LIN {X 0,Y 290.074,Z 393.623,A -85,B 0,C 180,E1 -16659.764,E2 -16659.764} C_VEL
LIN {X 0,Y 290.99,Z 387.907,A -85,B 0,C 180,E1 -16662.554,E2 -16662.554} C_VEL
LIN {X 0,Y 292.274,Z 381.468,A -85,B 0,C 180,E1 -16664.981,E2 -16664.981} C_VEL
LIN {X 0,Y 293.884,Z 373.47,A -85,B 0,C 180,E1 -16667.393,E2 -16667.393} C_VEL
LIN {X 0,Y 295.651,Z 365.107,A -85,B 0,C 180,E1 -16669.439,E2 -16669.439} C_VEL
LIN {X 0,Y 297.748,Z 355.042,A -85,B 0,C 180,E1 -16671.46,E2 -16671.46} C_VEL
LIN {X 0,Y 300.058,Z 343.813,A -85,B 0,C 180,E1 -16673.281,E2 -16673.281} C_VEL
LIN {X 0,Y 302.413,Z 331.182,A -85,B 0,C 180,E1 -16674.916,E2 -16674.916} C_VEL
LIN {X 0,Y 303.356,Z 325.276,A -85,B 0,C 180,E1 -16675.567,E2 -16675.567} C_VEL
LIN {X 0,Y 302.15,Z 313.202,A -85,B 0,C 180,E1 -16676.964,E2 -16676.964} C_VEL
LIN {X 0,Y 300.276,Z 302.153,A -85,B 0,C 180,E1 -16678.11,E2 -16678.11} C_VEL
LIN {X 0,Y 297.094,Z 288.461,A -85,B 0,C 180,E1 -16679.359,E2 -16679.359} C_VEL
LIN {X 0,Y 292.982,Z 275.551,A -85,B 0,C 180,E1 -16680.427,E2 -16680.427} C_VEL
LIN {X 0,Y 291.562,Z 271.297,A -85,B 0,C 180,E1 -16680.732,E2 -16680.732} C_VEL
LIN {X 0,Y 291.469,Z 270.609,A -85,B 0,C 180,E1 -16680.823,E2 -16680.823} C_VEL
LIN {X 0,Y 292.181,Z 265.371,A -85,B 0,C 180,E1 -16685.26,E2 -16685.26} C_VEL
LIN {X 0,Y 292.643,Z 261.551,A -85,B 0,C 180,E1 -16688.639,E2 -16688.639} C_VEL
LIN {X 0,Y 292.591,Z 258.142,A -85,B 0,C 180,E1 -16691.874,E2 -16691.874} C_VEL
LIN {X 0,Y 292.078,Z 254.325,A -85,B 0,C 180,E1 -16695.749,E2 -16695.749} C_VEL
LIN {X 0,Y 291.598,Z 250.967,A -85,B 0,C 180,E1 -16699.402,E2 -16699.402} C_VEL
LIN {X 0,Y 291.376,Z 249.818,A -85,B 0,C 180,E1 -16700.835,E2 -16700.835} C_VEL
LIN {X 0,Y 291.362,Z 249.821,A -85,B 0,C 180,E1 -16704.626,E2 -16704.626} C_VEL
LIN {X 0,Y 291.366,Z 249.819,A -85,B 0,C 180,E1 -16707.95,E2 -16707.95} C_VEL
LIN {X 0,Y 291.345,Z 249.821,A -85,B 0,C 180,E1 -16711.154,E2 -16711.154} C_VEL
LIN {X 0,Y 291.36,Z 249.818,A -85,B 0,C 180,E1 -16714.267,E2 -16714.267} C_VEL
LIN {X 0,Y 291.372,Z 249.817,A -85,B 0,C 180,E1 -16717.299,E2 -16717.299} C_VEL
LIN {X 0,Y 291.459,Z 249.806,A -85,B 0,C 180,E1 -16720.27,E2 -16720.27} C_VEL
LIN {X 0,Y 291.515,Z 249.797,A -85,B 0,C 180,E1 -16724.653,E2 -16724.653} C_VEL
LIN {X 0,Y 291.53,Z 249.79,A -85,B 0,C 180,E1 -16728.88,E2 -16728.88} C_VEL
LIN {X 0,Y 291.653,Z 249.782,A -85,B 0,C 180,E1 -16731.687,E2 -16731.687} C_VEL
LIN {X 0,Y 291.608,Z 249.785,A -85,B 0,C 180,E1 -16734.468,E2 -16734.468} C_VEL
LIN {X 0,Y 291.89,Z 249.751,A -85,B 0,C 180,E1 -16738.62,E2 -16738.62} C_VEL
LIN {X 0,Y 291.885,Z 249.752,A -85,B 0,C 180,E1 -16741.38,E2 -16741.38} C_VEL
LIN {X 0,Y 291.737,Z 249.77,A -85,B 0,C 180,E1 -16746.918,E2 -16746.918} C_VEL
LIN {X 0,Y 291.577,Z 249.791,A -85,B 0,C 180,E1 -16749.714,E2 -16749.714} C_VEL
LIN {X 0,Y 291.524,Z 249.795,A -85,B 0,C 180,E1 -16753.95,E2 -16753.95} C_VEL
LIN {X 0,Y 291.489,Z 249.801,A -85,B 0,C 180,E1 -16756.818,E2 -16756.818} C_VEL
LIN {X 0,Y 291.452,Z 249.804,A -85,B 0,C 180,E1 -16759.875,E2 -16759.875} C_VEL
LIN {X 0,Y 291.384,Z 249.814,A -85,B 0,C 180,E1 -16764.207,E2 -16764.207} C_VEL
LIN {X 0,Y 291.422,Z 249.81,A -85,B 0,C 180,E1 -16767.272,E2 -16767.272} C_VEL
LIN {X 0,Y 291.335,Z 249.821,A -85,B 0,C 180,E1 -16770.437,E2 -16770.437} C_VEL
LIN {X 0,Y 291.346,Z 249.82,A -85,B 0,C 180,E1 -16773.698,E2 -16773.698} C_VEL
LIN {X 0,Y 291.36,Z 249.818,A -85,B 0,C 180,E1 -16777.25,E2 -16777.25} C_VEL
LIN {X 0,Y 291.301,Z 249.828,A -85,B 0,C 180,E1 -16780.648,E2 -16780.648} C_VEL
LIN {X 0,Y 291.291,Z 249.828,A -85,B 0,C 180,E1 -16784.402,E2 -16784.402} C_VEL
LIN {X 0,Y 291.298,Z 249.899,A -85,B 0,C 180,E1 -16785.6,E2 -16785.6} C_VEL
LIN {X 0,Y 291.68,Z 252.914,A -85,B 0,C 180,E1 -16789.416,E2 -16789.416} C_VEL
LIN {X 0,Y 291.669,Z 255.712,A -85,B 0,C 180,E1 -16792.671,E2 -16792.671} C_VEL
LIN {X 0,Y 291.365,Z 258.994,A -85,B 0,C 180,E1 -16796.304,E2 -16796.304} C_VEL
LIN {X 0,Y 291.017,Z 261.76,A -85,B 0,C 180,E1 -16799.228,E2 -16799.228} C_VEL
LIN {X 0,Y 292.207,Z 265.24,A -85,B 0,C 180,E1 -16799.504,E2 -16799.504} C_VEL
LIN {X 0,Y 297.427,Z 279.57,A -85,B 0,C 180,E1 -16800.774,E2 -16800.774} C_VEL
LIN {X 0,Y 301.068,Z 292.825,A -85,B 0,C 180,E1 -16802.074,E2 -16802.074} C_VEL
LIN {X 0,Y 303.481,Z 304.486,A -85,B 0,C 180,E1 -16803.353,E2 -16803.353} C_VEL
LIN {X 0,Y 304.465,Z 311.537,A -85,B 0,C 180,E1 -16804.19,E2 -16804.19} C_VEL
LIN {X 0,Y 302.688,Z 323.224,A -85,B 0,C 180,E1 -16805.479,E2 -16805.479} C_VEL
LIN {X 0,Y 300.437,Z 335.236,A -85,B 0,C 180,E1 -16807.114,E2 -16807.114} C_VEL
LIN {X 0,Y 298.279,Z 346.061,A -85,B 0,C 180,E1 -16808.942,E2 -16808.942} C_VEL
LIN {X 0,Y 296.117,Z 355.805,A -85,B 0,C 180,E1 -16810.953,E2 -16810.953} C_VEL
LIN {X 0,Y 294.307,Z 363.822,A -85,B 0,C 180,E1 -16812.972,E2 -16812.972} C_VEL
LIN {X 0,Y 293,Z 370.611,A -85,B 0,C 180,E1 -16815.057,E2 -16815.057} C_VEL
LIN {X 0,Y 291.561,Z 377.013,A -85,B 0,C 180,E1 -16817.471,E2 -16817.471} C_VEL
LIN {X 0,Y 290.543,Z 382.685,A -85,B 0,C 180,E1 -16820.252,E2 -16820.252} C_VEL
LIN {X 0,Y 289.89,Z 386.805,A -85,B 0,C 180,E1 -16823.038,E2 -16823.038} C_VEL
LIN {X 0,Y 289.58,Z 389.498,A -85,B 0,C 180,E1 -16825.825,E2 -16825.825} C_VEL
LIN {X 0,Y 289.4,Z 390.846,A -85,B 0,C 180,E1 -16828.609,E2 -16828.609} C_VEL
LIN {X 0,Y 289.4,Z 390.876,A -85,B 0,C 180,E1 -16831.392,E2 -16831.392} C_VEL
LIN {X 0,Y 289.579,Z 389.585,A -85,B 0,C 180,E1 -16834.176,E2 -16834.176} C_VEL
LIN {X 0,Y 289.89,Z 386.945,A -85,B 0,C 180,E1 -16836.963,E2 -16836.963} C_VEL
LIN {X 0,Y 290.53,Z 382.885,A -85,B 0,C 180,E1 -16839.749,E2 -16839.749} C_VEL
LIN {X 0,Y 291.502,Z 377.275,A -85,B 0,C 180,E1 -16842.532,E2 -16842.532} C_VEL
LIN {X 0,Y 292.955,Z 370.934,A -85,B 0,C 180,E1 -16844.945,E2 -16844.945} C_VEL
LIN {X 0,Y 294.134,Z 364.631,A -85,B 0,C 180,E1 -16846.917,E2 -16846.917} C_VEL
LIN {X 0,Y 296.005,Z 356.282,A -85,B 0,C 180,E1 -16849.054,E2 -16849.054} C_VEL
LIN {X 0,Y 298.156,Z 346.631,A -85,B 0,C 180,E1 -16851.068,E2 -16851.068} C_VEL
LIN {X 0,Y 300.327,Z 335.919,A -85,B 0,C 180,E1 -16852.895,E2 -16852.895} C_VEL
LIN {X 0,Y 302.591,Z 324.044,A -85,B 0,C 180,E1 -16854.53,E2 -16854.53} C_VEL
LIN {X 0,Y 304.434,Z 312.231,A -85,B 0,C 180,E1 -16855.849,E2 -16855.849} C_VEL
LIN {X 0,Y 304.028,Z 307.686,A -85,B 0,C 180,E1 -16856.38,E2 -16856.38} C_VEL
LIN {X 0,Y 301.698,Z 295.36,A -85,B 0,C 180,E1 -16857.769,E2 -16857.769} C_VEL
LIN {X 0,Y 298.177,Z 281.925,A -85,B 0,C 180,E1 -16859.117,E2 -16859.117} C_VEL
LIN {X 0,Y 293.385,Z 268.223,A -85,B 0,C 180,E1 -16860.363,E2 -16860.363} C_VEL
LIN {X 0,Y 291.091,Z 262.196,A -85,B 0,C 180,E1 -16860.852,E2 -16860.852} C_VEL
LIN {X 0,Y 291.063,Z 261.708,A -85,B 0,C 180,E1 -16860.948,E2 -16860.948} C_VEL
LIN {X 0,Y 291.509,Z 257.962,A -85,B 0,C 180,E1 -16864.944,E2 -16864.944} C_VEL
LIN {X 0,Y 291.722,Z 254.552,A -85,B 0,C 180,E1 -16868.784,E2 -16868.784} C_VEL
LIN {X 0,Y 291.606,Z 252.15,A -85,B 0,C 180,E1 -16871.657,E2 -16871.657} C_VEL
LIN {X 0,Y 291.309,Z 250.01,A -85,B 0,C 180,E1 -16874.399,E2 -16874.399} C_VEL
LIN {X 0,Y 291.29,Z 249.83,A -85,B 0,C 180,E1 -16877.502,E2 -16877.502} C_VEL
LIN {X 0,Y 291.336,Z 249.822,A -85,B 0,C 180,E1 -16881.155,E2 -16881.155} C_VEL
LIN {X 0,Y 291.357,Z 249.82,A -85,B 0,C 180,E1 -16884.625,E2 -16884.625} C_VEL
LIN {X 0,Y 291.373,Z 249.816,A -85,B 0,C 180,E1 -16887.951,E2 -16887.951} C_VEL
LIN {X 0,Y 291.38,Z 249.816,A -85,B 0,C 180,E1 -16891.158,E2 -16891.158} C_VEL
LIN {X 0,Y 291.418,Z 249.806,A -85,B 0,C 180,E1 -16894.272,E2 -16894.272} C_VEL
LIN {X 0,Y 291.377,Z 249.816,A -85,B 0,C 180,E1 -16897.299,E2 -16897.299} C_VEL
LIN {X 0,Y 291.461,Z 249.804,A -85,B 0,C 180,E1 -16900.27,E2 -16900.27} C_VEL
LIN {X 0,Y 291.558,Z 249.791,A -85,B 0,C 180,E1 -16904.624,E2 -16904.624} C_VEL
LIN {X 0,Y 291.532,Z 249.795,A -85,B 0,C 180,E1 -16908.88,E2 -16908.88} C_VEL
LIN {X 0,Y 291.553,Z 249.792,A -85,B 0,C 180,E1 -16910.068,E2 -16910.068} C_VEL
LIN {X 0,Y 291.273,Z 249.832,A -85,B 0,C 180,E1 -16910.84,E2 -16910.84} C_VEL
LIN {X 0,Y 289.314,Z 250.08,A -85,B 0,C 180,E1 -16912.353,E2 -16912.353} C_VEL
LIN {X 0,Y 285.556,Z 250.544,A -85,B 0,C 180,E1 -16914.625,E2 -16914.625} C_VEL
LIN {X 0,Y 284.59,Z 250.661,A -85,B 0,C 180,E1 -16915.809,E2 -16915.809} C_VEL
LIN {X 0,Y 284.559,Z 250.662,A -85,B 0,C 180,E1 -16916.209,E2 -16916.209} C_VEL
LIN {X 0,Y 284.847,Z 250.63,A -85,B 0,C 180,E1 -16918.586,E2 -16918.586} C_VEL
LIN {X 0,Y 284.857,Z 250.628,A -85,B 0,C 180,E1 -16921.414,E2 -16921.414} C_VEL
LIN {X 0,Y 284.578,Z 250.661,A -85,B 0,C 180,E1 -16925.669,E2 -16925.669} C_VEL
LIN {X 0,Y 284.611,Z 250.658,A -85,B 0,C 180,E1 -16928.981,E2 -16928.981} C_VEL
LIN {X 0,Y 284.475,Z 250.675,A -85,B 0,C 180,E1 -16932.847,E2 -16932.847} C_VEL
LIN {X 0,Y 284.429,Z 250.682,A -85,B 0,C 180,E1 -16935.771,E2 -16935.771} C_VEL
LIN {X 0,Y 284.37,Z 250.688,A -85,B 0,C 180,E1 -16940.243,E2 -16940.243} C_VEL
LIN {X 0,Y 284.323,Z 250.694,A -85,B 0,C 180,E1 -16943.853,E2 -16943.853} C_VEL
LIN {X 0,Y 284.285,Z 250.698,A -85,B 0,C 180,E1 -16948.016,E2 -16948.016} C_VEL
LIN {X 0,Y 284.287,Z 250.696,A -85,B 0,C 180,E1 -16951.275,E2 -16951.275} C_VEL
LIN {X 0,Y 284.343,Z 250.696,A -85,B 0,C 180,E1 -16955.348,E2 -16955.348} C_VEL
LIN {X 0,Y 284.361,Z 250.857,A -85,B 0,C 180,E1 -16958.84,E2 -16958.84} C_VEL
LIN {X 0,Y 284.84,Z 253.775,A -85,B 0,C 180,E1 -16962.251,E2 -16962.251} C_VEL
LIN {X 0,Y 285.394,Z 257.638,A -85,B 0,C 180,E1 -16966.408,E2 -16966.408} C_VEL
LIN {X 0,Y 285.68,Z 260.917,A -85,B 0,C 180,E1 -16969.697,E2 -16969.697} C_VEL
LIN {X 0,Y 285.579,Z 263.394,A -85,B 0,C 180,E1 -16972.03,E2 -16972.03} C_VEL
LIN {X 0,Y 285.015,Z 267.188,A -85,B 0,C 180,E1 -16975.449,E2 -16975.449} C_VEL
LIN {X 0,Y 284.584,Z 270.583,A -85,B 0,C 180,E1 -16978.375,E2 -16978.375} C_VEL
LIN {X 0,Y 285.54,Z 273.818,A -85,B 0,C 180,E1 -16978.604,E2 -16978.604} C_VEL
LIN {X 0,Y 290.168,Z 287.833,A -85,B 0,C 180,E1 -16979.81,E2 -16979.81} C_VEL
LIN {X 0,Y 293.48,Z 301.655,A -85,B 0,C 180,E1 -16981.12,E2 -16981.12} C_VEL
LIN {X 0,Y 295.657,Z 314.286,A -85,B 0,C 180,E1 -16982.482,E2 -16982.482} C_VEL
LIN {X 0,Y 296.787,Z 325.408,A -85,B 0,C 180,E1 -16983.83,E2 -16983.83} C_VEL
LIN {X 0,Y 294.709,Z 338.214,A -85,B 0,C 180,E1 -16985.378,E2 -16985.378} C_VEL
LIN {X 0,Y 292.422,Z 349.218,A -85,B 0,C 180,E1 -16987.011,E2 -16987.011} C_VEL
LIN {X 0,Y 290.366,Z 358.608,A -85,B 0,C 180,E1 -16988.712,E2 -16988.712} C_VEL
LIN {X 0,Y 288.253,Z 368.057,A -85,B 0,C 180,E1 -16990.783,E2 -16990.783} C_VEL
LIN {X 0,Y 286.336,Z 376.898,A -85,B 0,C 180,E1 -16993.184,E2 -16993.184} C_VEL
LIN {X 0,Y 284.833,Z 384.342,A -85,B 0,C 180,E1 -16995.715,E2 -16995.715} C_VEL
LIN {X 0,Y 283.442,Z 390.884,A -85,B 0,C 180,E1 -16998.559,E2 -16998.559} C_VEL
LIN {X 0,Y 282.756,Z 395.785,A -85,B 0,C 180,E1 -17001.423,E2 -17001.423} C_VEL
LIN {X 0,Y 282.385,Z 399.194,A -85,B 0,C 180,E1 -17004.286,E2 -17004.286} C_VEL
LIN {X 0,Y 282.3,Z 401.211,A -85,B 0,C 180,E1 -17007.146,E2 -17007.146} C_VEL
LIN {X 0,Y 282.305,Z 401.876,A -85,B 0,C 180,E1 -17010,E2 -17010} C_VEL
LIN {X 0,Y 282.299,Z 401.199,A -85,B 0,C 180,E1 -17012.854,E2 -17012.854} C_VEL
LIN {X 0,Y 282.384,Z 399.173,A -85,B 0,C 180,E1 -17015.713,E2 -17015.713} C_VEL
LIN {X 0,Y 282.751,Z 395.752,A -85,B 0,C 180,E1 -17018.577,E2 -17018.577} C_VEL
LIN {X 0,Y 283.441,Z 390.832,A -85,B 0,C 180,E1 -17021.441,E2 -17021.441} C_VEL
LIN {X 0,Y 284.827,Z 384.277,A -85,B 0,C 180,E1 -17024.285,E2 -17024.285} C_VEL
LIN {X 0,Y 286.266,Z 376.973,A -85,B 0,C 180,E1 -17026.769,E2 -17026.769} C_VEL
LIN {X 0,Y 288.246,Z 367.95,A -85,B 0,C 180,E1 -17029.218,E2 -17029.218} C_VEL
LIN {X 0,Y 290.355,Z 358.477,A -85,B 0,C 180,E1 -17031.289,E2 -17031.289} C_VEL
LIN {X 0,Y 292.637,Z 347.993,A -85,B 0,C 180,E1 -17033.158,E2 -17033.158} C_VEL
LIN {X 0,Y 294.942,Z 336.425,A -85,B 0,C 180,E1 -17034.833,E2 -17034.833} C_VEL
LIN {X 0,Y 296.701,Z 326.763,A -85,B 0,C 180,E1 -17035.989,E2 -17035.989} C_VEL
LIN {X 0,Y 295.956,Z 317.316,A -85,B 0,C 180,E1 -17037.14,E2 -17037.14} C_VEL
LIN {X 0,Y 294.394,Z 306.593,A -85,B 0,C 180,E1 -17038.335,E2 -17038.335} C_VEL
LIN {X 0,Y 291.364,Z 292.508,A -85,B 0,C 180,E1 -17039.732,E2 -17039.732} C_VEL
LIN {X 0,Y 287.7,Z 280.05,A -85,B 0,C 180,E1 -17040.844,E2 -17040.844} C_VEL
LIN {X 0,Y 284.725,Z 271.673,A -85,B 0,C 180,E1 -17041.534,E2 -17041.534} C_VEL
LIN {X 0,Y 284.549,Z 270.482,A -85,B 0,C 180,E1 -17041.634,E2 -17041.634} C_VEL
LIN {X 0,Y 285.183,Z 265.952,A -85,B 0,C 180,E1 -17045.586,E2 -17045.586} C_VEL
LIN {X 0,Y 285.55,Z 263.251,A -85,B 0,C 180,E1 -17048.039,E2 -17048.039} C_VEL
LIN {X 0,Y 285.67,Z 260.868,A -85,B 0,C 180,E1 -17050.301,E2 -17050.301} C_VEL
LIN {X 0,Y 285.367,Z 257.593,A -85,B 0,C 180,E1 -17053.597,E2 -17053.597} C_VEL
LIN {X 0,Y 284.839,Z 253.727,A -85,B 0,C 180,E1 -17057.749,E2 -17057.749} C_VEL
LIN {X 0,Y 284.328,Z 250.696,A -85,B 0,C 180,E1 -17061.382,E2 -17061.382} C_VEL
LIN {X 0,Y 284.309,Z 250.7,A -85,B 0,C 180,E1 -17065.351,E2 -17065.351} C_VEL
LIN {X 0,Y 284.285,Z 250.701,A -85,B 0,C 180,E1 -17068.725,E2 -17068.725} C_VEL
LIN {X 0,Y 284.284,Z 250.7,A -85,B 0,C 180,E1 -17071.984,E2 -17071.984} C_VEL
LIN {X 0,Y 284.322,Z 250.695,A -85,B 0,C 180,E1 -17076.147,E2 -17076.147} C_VEL
LIN {X 0,Y 284.377,Z 250.687,A -85,B 0,C 180,E1 -17079.904,E2 -17079.904} C_VEL
LIN {X 0,Y 284.455,Z 250.677,A -85,B 0,C 180,E1 -17084.487,E2 -17084.487} C_VEL
LIN {X 0,Y 284.484,Z 250.67,A -85,B 0,C 180,E1 -17088.601,E2 -17088.601} C_VEL
LIN {X 0,Y 284.61,Z 250.658,A -85,B 0,C 180,E1 -17091.48,E2 -17091.48} C_VEL
LIN {X 0,Y 284.577,Z 250.661,A -85,B 0,C 180,E1 -17094.331,E2 -17094.331} C_VEL
LIN {X 0,Y 284.856,Z 250.627,A -85,B 0,C 180,E1 -17098.586,E2 -17098.586} C_VEL
LIN {X 0,Y 284.852,Z 250.628,A -85,B 0,C 180,E1 -17101.414,E2 -17101.414} C_VEL
LIN {X 0,Y 284.688,Z 250.648,A -85,B 0,C 180,E1 -17107.09,E2 -17107.09} C_VEL
LIN {X 0,Y 284.521,Z 250.671,A -85,B 0,C 180,E1 -17109.957,E2 -17109.957} C_VEL
LIN {X 0,Y 284.483,Z 250.673,A -85,B 0,C 180,E1 -17114.303,E2 -17114.303} C_VEL
LIN {X 0,Y 284.427,Z 250.681,A -85,B 0,C 180,E1 -17117.248,E2 -17117.248} C_VEL
LIN {X 0,Y 284.379,Z 250.685,A -85,B 0,C 180,E1 -17120.242,E2 -17120.242} C_VEL
LIN {X 0,Y 284.34,Z 250.691,A -85,B 0,C 180,E1 -17124.847,E2 -17124.847} C_VEL
LIN {X 0,Y 284.33,Z 250.693,A -85,B 0,C 180,E1 -17128.011,E2 -17128.011} C_VEL
LIN {X 0,Y 284.295,Z 250.697,A -85,B 0,C 180,E1 -17131.275,E2 -17131.275} C_VEL
LIN {X 0,Y 284.337,Z 250.693,A -85,B 0,C 180,E1 -17135.347,E2 -17135.347} C_VEL
LIN {X 0,Y 284.299,Z 250.697,A -85,B 0,C 180,E1 -17138.171,E2 -17138.171} C_VEL
LIN {X 0,Y 284.238,Z 250.706,A -85,B 0,C 180,E1 -17142.117,E2 -17142.117} C_VEL
LIN {X 0,Y 284.247,Z 250.706,A -85,B 0,C 180,E1 -17144.191,E2 -17144.191} C_VEL
LIN {X 0,Y 284.38,Z 251.545,A -85,B 0,C 180,E1 -17146.213,E2 -17146.213} C_VEL
LIN {X 0,Y 284.595,Z 253.063,A -85,B 0,C 180,E1 -17148.183,E2 -17148.183} C_VEL
LIN {X 0,Y 284.701,Z 254.568,A -85,B 0,C 180,E1 -17150.072,E2 -17150.072} C_VEL
LIN {X 0,Y 284.568,Z 257.626,A -85,B 0,C 180,E1 -17153.649,E2 -17153.649} C_VEL
LIN {X 0,Y 284.23,Z 260.816,A -85,B 0,C 180,E1 -17157.214,E2 -17157.214} C_VEL
LIN {X 0,Y 284.093,Z 261.908,A -85,B 0,C 180,E1 -17158.4,E2 -17158.4} C_VEL
LIN {X 0,Y 285.117,Z 265.123,A -85,B 0,C 180,E1 -17158.651,E2 -17158.651} C_VEL
LIN {X 0,Y 290.208,Z 278.632,A -85,B 0,C 180,E1 -17159.911,E2 -17159.911} C_VEL
LIN {X 0,Y 293.978,Z 291.63,A -85,B 0,C 180,E1 -17161.232,E2 -17161.232} C_VEL
LIN {X 0,Y 296.699,Z 304.155,A -85,B 0,C 180,E1 -17162.647,E2 -17162.647} C_VEL
LIN {X 0,Y 297.909,Z 312.67,A -85,B 0,C 180,E1 -17163.697,E2 -17163.697} C_VEL
LIN {X 0,Y 296.004,Z 324.651,A -85,B 0,C 180,E1 -17165.075,E2 -17165.075} C_VEL
LIN {X 0,Y 293.68,Z 336.441,A -85,B 0,C 180,E1 -17166.743,E2 -17166.743} C_VEL
LIN {X 0,Y 291.627,Z 346.2,A -85,B 0,C 180,E1 -17168.438,E2 -17168.438} C_VEL
LIN {X 0,Y 289.411,Z 355.942,A -85,B 0,C 180,E1 -17170.494,E2 -17170.494} C_VEL
LIN {X 0,Y 287.391,Z 364.434,A -85,B 0,C 180,E1 -17172.692,E2 -17172.692} C_VEL
LIN {X 0,Y 286.13,Z 370.747,A -85,B 0,C 180,E1 -17174.69,E2 -17174.69} C_VEL
LIN {X 0,Y 284.595,Z 377.15,A -85,B 0,C 180,E1 -17177.159,E2 -17177.159} C_VEL
LIN {X 0,Y 283.515,Z 382.822,A -85,B 0,C 180,E1 -17180.007,E2 -17180.007} C_VEL
LIN {X 0,Y 282.836,Z 386.941,A -85,B 0,C 180,E1 -17182.863,E2 -17182.863} C_VEL
LIN {X 0,Y 282.486,Z 389.633,A -85,B 0,C 180,E1 -17185.72,E2 -17185.72} C_VEL
LIN {X 0,Y 282.326,Z 390.98,A -85,B 0,C 180,E1 -17188.574,E2 -17188.574} C_VEL
LIN {X 0,Y 282.326,Z 391.01,A -85,B 0,C 180,E1 -17191.427,E2 -17191.427} C_VEL
LIN {X 0,Y 282.486,Z 389.72,A -85,B 0,C 180,E1 -17194.281,E2 -17194.281} C_VEL
LIN {X 0,Y 282.836,Z 387.079,A -85,B 0,C 180,E1 -17197.137,E2 -17197.137} C_VEL
LIN {X 0,Y 283.5,Z 383.019,A -85,B 0,C 180,E1 -17199.993,E2 -17199.993} C_VEL
LIN {X 0,Y 284.54,Z 377.409,A -85,B 0,C 180,E1 -17202.844,E2 -17202.844} C_VEL
LIN {X 0,Y 286.096,Z 371.067,A -85,B 0,C 180,E1 -17205.312,E2 -17205.312} C_VEL
LIN {X 0,Y 287.477,Z 363.995,A -85,B 0,C 180,E1 -17207.552,E2 -17207.552} C_VEL
LIN {X 0,Y 289.645,Z 354.934,A -85,B 0,C 180,E1 -17209.859,E2 -17209.859} C_VEL
LIN {X 0,Y 291.926,Z 344.987,A -85,B 0,C 180,E1 -17211.911,E2 -17211.911} C_VEL
LIN {X 0,Y 294.28,Z 333.911,A -85,B 0,C 180,E1 -17213.767,E2 -17213.767} C_VEL
LIN {X 0,Y 296.409,Z 322.879,A -85,B 0,C 180,E1 -17215.264,E2 -17215.264} C_VEL
LIN {X 0,Y 297.952,Z 312.708,A -85,B 0,C 180,E1 -17216.413,E2 -17216.413} C_VEL
LIN {X 0,Y 296.102,Z 300.857,A -85,B 0,C 180,E1 -17217.855,E2 -17217.855} C_VEL
LIN {X 0,Y 293.155,Z 288.434,A -85,B 0,C 180,E1 -17219.223,E2 -17219.223} C_VEL
LIN {X 0,Y 289.519,Z 276.682,A -85,B 0,C 180,E1 -17220.401,E2 -17220.401} C_VEL
LIN {X 0,Y 285.037,Z 264.924,A -85,B 0,C 180,E1 -17221.491,E2 -17221.491} C_VEL
LIN {X 0,Y 284.116,Z 261.905,A -85,B 0,C 180,E1 -17221.729,E2 -17221.729} C_VEL
LIN {X 0,Y 284.508,Z 258.59,A -85,B 0,C 180,E1 -17225.395,E2 -17225.395} C_VEL
LIN {X 0,Y 284.669,Z 256.208,A -85,B 0,C 180,E1 -17228.113,E2 -17228.113} C_VEL
LIN {X 0,Y 284.68,Z 254.573,A -85,B 0,C 180,E1 -17230.065,E2 -17230.065} C_VEL
LIN {X 0,Y 284.561,Z 252.884,A -85,B 0,C 180,E1 -17232.189,E2 -17232.189} C_VEL
LIN {X 0,Y 284.346,Z 251.335,A -85,B 0,C 180,E1 -17234.211,E2 -17234.211} C_VEL
LIN {X 0,Y 284.257,Z 250.707,A -85,B 0,C 180,E1 -17236.189,E2 -17236.189} C_VEL
LIN {X 0,Y 284.285,Z 250.699,A -85,B 0,C 180,E1 -17240.03,E2 -17240.03} C_VEL
LIN {X 0,Y 284.323,Z 250.695,A -85,B 0,C 180,E1 -17243.612,E2 -17243.612} C_VEL
LIN {X 0,Y 284.31,Z 250.696,A -85,B 0,C 180,E1 -17247.19,E2 -17247.19} C_VEL
LIN {X 0,Y 284.358,Z 250.69,A -85,B 0,C 180,E1 -17250.376,E2 -17250.376} C_VEL
LIN {X 0,Y 284.38,Z 250.687,A -85,B 0,C 180,E1 -17253.587,E2 -17253.587} C_VEL
LIN {X 0,Y 284.336,Z 250.692,A -85,B 0,C 180,E1 -17256.704,E2 -17256.704} C_VEL
LIN {X 0,Y 284.406,Z 250.683,A -85,B 0,C 180,E1 -17261.262,E2 -17261.262} C_VEL
LIN {X 0,Y 284.495,Z 250.671,A -85,B 0,C 180,E1 -17264.459,E2 -17264.459} C_VEL
LIN {X 0,Y 284.486,Z 250.674,A -85,B 0,C 180,E1 -17268.601,E2 -17268.601} C_VEL
LIN {X 0,Y 284.625,Z 250.656,A -85,B 0,C 180,E1 -17271.48,E2 -17271.48} C_VEL
LIN {X 0,Y 284.593,Z 250.658,A -85,B 0,C 180,E1 -17274.331,E2 -17274.331} C_VEL
LIN {X 0,Y 284.559,Z 250.662,A -85,B 0,C 180,E1 -17276.209,E2 -17276.209} C_VEL
LIN {X 0,Y 284.041,Z 250.727,A -85,B 0,C 180,E1 -17277.393,E2 -17277.393} C_VEL
LIN {X 0,Y 281.31,Z 251.068,A -85,B 0,C 180,E1 -17279.323,E2 -17279.323} C_VEL
LIN {X 0,Y 278.892,Z 251.37,A -85,B 0,C 180,E1 -17280.891,E2 -17280.891} C_VEL
LIN {X 0,Y 277.817,Z 251.502,A -85,B 0,C 180,E1 -17282.104,E2 -17282.104} C_VEL
LIN {X 0,Y 277.714,Z 251.514,A -85,B 0,C 180,E1 -17282.516,E2 -17282.516} C_VEL
LIN {X 0,Y 277.604,Z 251.529,A -85,B 0,C 180,E1 -17287.272,E2 -17287.272} C_VEL
LIN {X 0,Y 277.46,Z 251.549,A -85,B 0,C 180,E1 -17290.213,E2 -17290.213} C_VEL
LIN {X 0,Y 277.417,Z 251.555,A -85,B 0,C 180,E1 -17294.675,E2 -17294.675} C_VEL
LIN {X 0,Y 277.331,Z 251.564,A -85,B 0,C 180,E1 -17299.235,E2 -17299.235} C_VEL
LIN {X 0,Y 277.284,Z 251.571,A -85,B 0,C 180,E1 -17303.924,E2 -17303.924} C_VEL
LIN {X 0,Y 277.271,Z 251.573,A -85,B 0,C 180,E1 -17307.483,E2 -17307.483} C_VEL
LIN {X 0,Y 277.249,Z 251.576,A -85,B 0,C 180,E1 -17310.472,E2 -17310.472} C_VEL
LIN {X 0,Y 277.248,Z 251.576,A -85,B 0,C 180,E1 -17313.896,E2 -17313.896} C_VEL
LIN {X 0,Y 277.283,Z 251.574,A -85,B 0,C 180,E1 -17318.027,E2 -17318.027} C_VEL
LIN {X 0,Y 277.711,Z 254.115,A -85,B 0,C 180,E1 -17321.146,E2 -17321.146} C_VEL
LIN {X 0,Y 278.214,Z 257.527,A -85,B 0,C 180,E1 -17325.017,E2 -17325.017} C_VEL
LIN {X 0,Y 278.473,Z 259.407,A -85,B 0,C 180,E1 -17327.045,E2 -17327.045} C_VEL
LIN {X 0,Y 278.62,Z 261.469,A -85,B 0,C 180,E1 -17329.177,E2 -17329.177} C_VEL
LIN {X 0,Y 278.577,Z 263.807,A -85,B 0,C 180,E1 -17331.451,E2 -17331.451} C_VEL
LIN {X 0,Y 278.132,Z 267.058,A -85,B 0,C 180,E1 -17334.466,E2 -17334.466} C_VEL
LIN {X 0,Y 277.672,Z 270.398,A -85,B 0,C 180,E1 -17337.481,E2 -17337.481} C_VEL
LIN {X 0,Y 278.713,Z 273.807,A -85,B 0,C 180,E1 -17337.747,E2 -17337.747} C_VEL
LIN {X 0,Y 283.181,Z 287.194,A -85,B 0,C 180,E1 -17338.956,E2 -17338.956} C_VEL
LIN {X 0,Y 285.98,Z 298.051,A -85,B 0,C 180,E1 -17340.02,E2 -17340.02} C_VEL
LIN {X 0,Y 288.453,Z 310.929,A -85,B 0,C 180,E1 -17341.415,E2 -17341.415} C_VEL
LIN {X 0,Y 289.85,Z 322.084,A -85,B 0,C 180,E1 -17342.764,E2 -17342.764} C_VEL
LIN {X 0,Y 290.205,Z 326.857,A -85,B 0,C 180,E1 -17343.384,E2 -17343.384} C_VEL
LIN {X 0,Y 287.959,Z 339.465,A -85,B 0,C 180,E1 -17344.982,E2 -17344.982} C_VEL
LIN {X 0,Y 285.391,Z 351.054,A -85,B 0,C 180,E1 -17346.795,E2 -17346.795} C_VEL
LIN {X 0,Y 282.926,Z 361.793,A -85,B 0,C 180,E1 -17348.888,E2 -17348.888} C_VEL
LIN {X 0,Y 280.867,Z 370.664,A -85,B 0,C 180,E1 -17351.016,E2 -17351.016} C_VEL
LIN {X 0,Y 279.005,Z 379.271,A -85,B 0,C 180,E1 -17353.572,E2 -17353.572} C_VEL
LIN {X 0,Y 277.487,Z 386.025,A -85,B 0,C 180,E1 -17356.077,E2 -17356.077} C_VEL
LIN {X 0,Y 276.432,Z 390.749,A -85,B 0,C 180,E1 -17358.264,E2 -17358.264} C_VEL
LIN {X 0,Y 275.692,Z 395.651,A -85,B 0,C 180,E1 -17361.202,E2 -17361.202} C_VEL
LIN {X 0,Y 275.296,Z 399.06,A -85,B 0,C 180,E1 -17364.139,E2 -17364.139} C_VEL
LIN {X 0,Y 275.212,Z 401.076,A -85,B 0,C 180,E1 -17367.072,E2 -17367.072} C_VEL
LIN {X 0,Y 275.229,Z 401.741,A -85,B 0,C 180,E1 -17370,E2 -17370} C_VEL
LIN {X 0,Y 275.211,Z 401.064,A -85,B 0,C 180,E1 -17372.927,E2 -17372.927} C_VEL
LIN {X 0,Y 275.296,Z 399.038,A -85,B 0,C 180,E1 -17375.861,E2 -17375.861} C_VEL
LIN {X 0,Y 275.688,Z 395.615,A -85,B 0,C 180,E1 -17378.798,E2 -17378.798} C_VEL
LIN {X 0,Y 276.431,Z 390.695,A -85,B 0,C 180,E1 -17381.735,E2 -17381.735} C_VEL
LIN {X 0,Y 277.887,Z 384.14,A -85,B 0,C 180,E1 -17384.65,E2 -17384.65} C_VEL
LIN {X 0,Y 279.279,Z 377.41,A -85,B 0,C 180,E1 -17387.008,E2 -17387.008} C_VEL
LIN {X 0,Y 281.163,Z 369.202,A -85,B 0,C 180,E1 -17389.342,E2 -17389.342} C_VEL
LIN {X 0,Y 283.324,Z 360.038,A -85,B 0,C 180,E1 -17391.462,E2 -17391.462} C_VEL
LIN {X 0,Y 285.393,Z 350.903,A -85,B 0,C 180,E1 -17393.204,E2 -17393.204} C_VEL
LIN {X 0,Y 287.991,Z 339.052,A -85,B 0,C 180,E1 -17395.052,E2 -17395.052} C_VEL
LIN {X 0,Y 290.178,Z 326.62,A -85,B 0,C 180,E1 -17396.619,E2 -17396.619} C_VEL
LIN {X 0,Y 288.885,Z 313.708,A -85,B 0,C 180,E1 -17398.231,E2 -17398.231} C_VEL
LIN {X 0,Y 286.496,Z 300.517,A -85,B 0,C 180,E1 -17399.695,E2 -17399.695} C_VEL
LIN {X 0,Y 283.194,Z 287.173,A -85,B 0,C 180,E1 -17401.008,E2 -17401.008} C_VEL
LIN {X 0,Y 278.532,Z 273.465,A -85,B 0,C 180,E1 -17402.25,E2 -17402.25} C_VEL
LIN {X 0,Y 277.645,Z 270.372,A -85,B 0,C 180,E1 -17402.488,E2 -17402.488} C_VEL
LIN {X 0,Y 278.223,Z 266.399,A -85,B 0,C 180,E1 -17406.067,E2 -17406.067} C_VEL
LIN {X 0,Y 278.586,Z 263.19,A -85,B 0,C 180,E1 -17409.101,E2 -17409.101} C_VEL
LIN {X 0,Y 278.602,Z 261.265,A -85,B 0,C 180,E1 -17410.986,E2 -17410.986} C_VEL
LIN {X 0,Y 278.339,Z 258.398,A -85,B 0,C 180,E1 -17413.986,E2 -17413.986} C_VEL
LIN {X 0,Y 277.901,Z 255.521,A -85,B 0,C 180,E1 -17417.172,E2 -17417.172} C_VEL
LIN {X 0,Y 277.426,Z 252.53,A -85,B 0,C 180,E1 -17420.704,E2 -17420.704} C_VEL
LIN {X 0,Y 277.302,Z 251.572,A -85,B 0,C 180,E1 -17422.162,E2 -17422.162} C_VEL
LIN {X 0,Y 277.247,Z 251.579,A -85,B 0,C 180,E1 -17426.104,E2 -17426.104} C_VEL
LIN {X 0,Y 277.262,Z 251.575,A -85,B 0,C 180,E1 -17429.539,E2 -17429.539} C_VEL
LIN {X 0,Y 277.293,Z 251.57,A -85,B 0,C 180,E1 -17432.857,E2 -17432.857} C_VEL
LIN {X 0,Y 277.283,Z 251.572,A -85,B 0,C 180,E1 -17436.075,E2 -17436.075} C_VEL
LIN {X 0,Y 277.33,Z 251.566,A -85,B 0,C 180,E1 -17440.765,E2 -17440.765} C_VEL
LIN {X 0,Y 277.416,Z 251.55,A -85,B 0,C 180,E1 -17445.325,E2 -17445.325} C_VEL
LIN {X 0,Y 277.458,Z 251.542,A -85,B 0,C 180,E1 -17449.787,E2 -17449.787} C_VEL
LIN {X 0,Y 277.603,Z 251.529,A -85,B 0,C 180,E1 -17452.728,E2 -17452.728} C_VEL
LIN {X 0,Y 277.822,Z 251.504,A -85,B 0,C 180,E1 -17458.551,E2 -17458.551} C_VEL
LIN {X 0,Y 277.818,Z 251.504,A -85,B 0,C 180,E1 -17461.45,E2 -17461.45} C_VEL
LIN {X 0,Y 277.642,Z 251.525,A -85,B 0,C 180,E1 -17467.271,E2 -17467.271} C_VEL
LIN {X 0,Y 277.463,Z 251.549,A -85,B 0,C 180,E1 -17470.213,E2 -17470.213} C_VEL
LIN {X 0,Y 277.436,Z 251.553,A -85,B 0,C 180,E1 -17474.674,E2 -17474.674} C_VEL
LIN {X 0,Y 277.346,Z 251.564,A -85,B 0,C 180,E1 -17479.234,E2 -17479.234} C_VEL
LIN {X 0,Y 277.293,Z 251.569,A -85,B 0,C 180,E1 -17484.158,E2 -17484.158} C_VEL
LIN {X 0,Y 277.326,Z 251.565,A -85,B 0,C 180,E1 -17487.505,E2 -17487.505} C_VEL
LIN {X 0,Y 277.273,Z 251.572,A -85,B 0,C 180,E1 -17490.481,E2 -17490.481} C_VEL
LIN {X 0,Y 277.247,Z 251.576,A -85,B 0,C 180,E1 -17493.896,E2 -17493.896} C_VEL
LIN {X 0,Y 277.256,Z 251.576,A -85,B 0,C 180,E1 -17497.471,E2 -17497.471} C_VEL
LIN {X 0,Y 277.185,Z 251.585,A -85,B 0,C 180,E1 -17501.241,E2 -17501.241} C_VEL
LIN {X 0,Y 277.225,Z 251.695,A -85,B 0,C 180,E1 -17504.779,E2 -17504.779} C_VEL
LIN {X 0,Y 277.606,Z 254.725,A -85,B 0,C 180,E1 -17508.835,E2 -17508.835} C_VEL
LIN {X 0,Y 277.607,Z 257.751,A -85,B 0,C 180,E1 -17512.584,E2 -17512.584} C_VEL
LIN {X 0,Y 277.281,Z 260.823,A -85,B 0,C 180,E1 -17516.109,E2 -17516.109} C_VEL
LIN {X 0,Y 277.164,Z 262.065,A -85,B 0,C 180,E1 -17517.517,E2 -17517.517} C_VEL
LIN {X 0,Y 278.361,Z 265.521,A -85,B 0,C 180,E1 -17517.808,E2 -17517.808} C_VEL
LIN {X 0,Y 283.194,Z 278.383,A -85,B 0,C 180,E1 -17519.062,E2 -17519.062} C_VEL
LIN {X 0,Y 286.972,Z 290.893,A -85,B 0,C 180,E1 -17520.391,E2 -17520.391} C_VEL
LIN {X 0,Y 289.722,Z 303.061,A -85,B 0,C 180,E1 -17521.806,E2 -17521.806} C_VEL
LIN {X 0,Y 291.381,Z 313.78,A -85,B 0,C 180,E1 -17523.18,E2 -17523.18} C_VEL
LIN {X 0,Y 289.333,Z 326.078,A -85,B 0,C 180,E1 -17524.652,E2 -17524.652} C_VEL
LIN {X 0,Y 286.939,Z 337.646,A -85,B 0,C 180,E1 -17526.355,E2 -17526.355} C_VEL
LIN {X 0,Y 284.658,Z 348.113,A -85,B 0,C 180,E1 -17528.264,E2 -17528.264} C_VEL
LIN {X 0,Y 282.333,Z 357.56,A -85,B 0,C 180,E1 -17530.364,E2 -17530.364} C_VEL
LIN {X 0,Y 280.412,Z 365.385,A -85,B 0,C 180,E1 -17532.497,E2 -17532.497} C_VEL
LIN {X 0,Y 279.033,Z 371.886,A -85,B 0,C 180,E1 -17534.665,E2 -17534.665} C_VEL
LIN {X 0,Y 277.644,Z 377.287,A -85,B 0,C 180,E1 -17536.832,E2 -17536.832} C_VEL
LIN {X 0,Y 276.499,Z 382.958,A -85,B 0,C 180,E1 -17539.751,E2 -17539.751} C_VEL
LIN {X 0,Y 275.779,Z 387.077,A -85,B 0,C 180,E1 -17542.68,E2 -17542.68} C_VEL
LIN {X 0,Y 275.398,Z 389.768,A -85,B 0,C 180,E1 -17545.609,E2 -17545.609} C_VEL
LIN {X 0,Y 275.253,Z 391.115,A -85,B 0,C 180,E1 -17548.537,E2 -17548.537} C_VEL
LIN {X 0,Y 275.253,Z 391.144,A -85,B 0,C 180,E1 -17551.463,E2 -17551.463} C_VEL
LIN {X 0,Y 275.396,Z 389.854,A -85,B 0,C 180,E1 -17554.391,E2 -17554.391} C_VEL
LIN {X 0,Y 275.779,Z 387.213,A -85,B 0,C 180,E1 -17557.321,E2 -17557.321} C_VEL
LIN {X 0,Y 276.483,Z 383.153,A -85,B 0,C 180,E1 -17560.25,E2 -17560.25} C_VEL
LIN {X 0,Y 277.592,Z 377.543,A -85,B 0,C 180,E1 -17563.171,E2 -17563.171} C_VEL
LIN {X 0,Y 279.251,Z 371.2,A -85,B 0,C 180,E1 -17565.697,E2 -17565.697} C_VEL
LIN {X 0,Y 280.897,Z 363.323,A -85,B 0,C 180,E1 -17568.224,E2 -17568.224} C_VEL
LIN {X 0,Y 282.968,Z 355.066,A -85,B 0,C 180,E1 -17570.348,E2 -17570.348} C_VEL
LIN {X 0,Y 285.323,Z 345.119,A -85,B 0,C 180,E1 -17572.445,E2 -17572.445} C_VEL
LIN {X 0,Y 287.795,Z 334.042,A -85,B 0,C 180,E1 -17574.336,E2 -17574.336} C_VEL
LIN {X 0,Y 290.009,Z 323.009,A -85,B 0,C 180,E1 -17575.862,E2 -17575.862} C_VEL
LIN {X 0,Y 291.411,Z 314.188,A -85,B 0,C 180,E1 -17576.887,E2 -17576.887} C_VEL
LIN {X 0,Y 289.624,Z 302.329,A -85,B 0,C 180,E1 -17578.4,E2 -17578.4} C_VEL
LIN {X 0,Y 286.55,Z 289.093,A -85,B 0,C 180,E1 -17579.924,E2 -17579.924} C_VEL
LIN {X 0,Y 282.444,Z 276.085,A -85,B 0,C 180,E1 -17581.289,E2 -17581.289} C_VEL
LIN {X 0,Y 277.388,Z 263.166,A -85,B 0,C 180,E1 -17582.533,E2 -17582.533} C_VEL
LIN {X 0,Y 277.194,Z 262.058,A -85,B 0,C 180,E1 -17582.618,E2 -17582.618} C_VEL
LIN {X 0,Y 277.511,Z 259.196,A -85,B 0,C 180,E1 -17585.864,E2 -17585.864} C_VEL
LIN {X 0,Y 277.643,Z 256.354,A -85,B 0,C 180,E1 -17589.259,E2 -17589.259} C_VEL
LIN {X 0,Y 277.486,Z 253.628,A -85,B 0,C 180,E1 -17592.735,E2 -17592.735} C_VEL
LIN {X 0,Y 277.228,Z 251.8,A -85,B 0,C 180,E1 -17595.221,E2 -17595.221} C_VEL
LIN {X 0,Y 277.186,Z 251.585,A -85,B 0,C 180,E1 -17598.759,E2 -17598.759} C_VEL
LIN {X 0,Y 277.257,Z 251.576,A -85,B 0,C 180,E1 -17602.529,E2 -17602.529} C_VEL
LIN {X 0,Y 277.248,Z 251.577,A -85,B 0,C 180,E1 -17606.104,E2 -17606.104} C_VEL
LIN {X 0,Y 277.264,Z 251.574,A -85,B 0,C 180,E1 -17609.539,E2 -17609.539} C_VEL
LIN {X 0,Y 277.361,Z 251.562,A -85,B 0,C 180,E1 -17612.864,E2 -17612.864} C_VEL
LIN {X 0,Y 277.3,Z 251.568,A -85,B 0,C 180,E1 -17616.077,E2 -17616.077} C_VEL
LIN {X 0,Y 277.347,Z 251.564,A -85,B 0,C 180,E1 -17620.766,E2 -17620.766} C_VEL
LIN {X 0,Y 277.438,Z 251.552,A -85,B 0,C 180,E1 -17625.326,E2 -17625.326} C_VEL
LIN {X 0,Y 277.46,Z 251.547,A -85,B 0,C 180,E1 -17629.787,E2 -17629.787} C_VEL
LIN {X 0,Y 277.631,Z 251.527,A -85,B 0,C 180,E1 -17632.728,E2 -17632.728} C_VEL
LIN {X 0,Y 277.814,Z 251.506,A -85,B 0,C 180,E1 -17638.55,E2 -17638.55} C_VEL
LIN {X 0,Y 277.823,Z 251.505,A -85,B 0,C 180,E1 -17641.449,E2 -17641.449} C_VEL
LIN {X 0,Y 277.714,Z 251.514,A -85,B 0,C 180,E1 -17642.516,E2 -17642.516} C_VEL
LIN {X 0,Y 276.987,Z 251.608,A -85,B 0,C 180,E1 -17643.724,E2 -17643.724} C_VEL
LIN {X 0,Y 274.056,Z 251.972,A -85,B 0,C 180,E1 -17645.692,E2 -17645.692} C_VEL
LIN {X 0,Y 271.614,Z 252.275,A -85,B 0,C 180,E1 -17647.291,E2 -17647.291} C_VEL
LIN {X 0,Y 270.597,Z 252.405,A -85,B 0,C 180,E1 -17648.532,E2 -17648.532} C_VEL
LIN {X 0,Y 270.529,Z 252.412,A -85,B 0,C 180,E1 -17648.952,E2 -17648.952} C_VEL
LIN {X 0,Y 270.352,Z 252.435,A -85,B 0,C 180,E1 -17653.53,E2 -17653.53} C_VEL
LIN {X 0,Y 270.293,Z 252.441,A -85,B 0,C 180,E1 -17656.619,E2 -17656.619} C_VEL
LIN {X 0,Y 270.274,Z 252.444,A -85,B 0,C 180,E1 -17660.59,E2 -17660.59} C_VEL
LIN {X 0,Y 270.226,Z 252.447,A -85,B 0,C 180,E1 -17664.59,E2 -17664.59} C_VEL
LIN {X 0,Y 270.2,Z 252.452,A -85,B 0,C 180,E1 -17667.917,E2 -17667.917} C_VEL
LIN {X 0,Y 270.175,Z 252.453,A -85,B 0,C 180,E1 -17671.349,E2 -17671.349} C_VEL
LIN {X 0,Y 270.203,Z 252.457,A -85,B 0,C 180,E1 -17674.905,E2 -17674.905} C_VEL
LIN {X 0,Y 270.273,Z 252.634,A -85,B 0,C 180,E1 -17677.667,E2 -17677.667} C_VEL
LIN {X 0,Y 270.737,Z 255.421,A -85,B 0,C 180,E1 -17681.166,E2 -17681.166} C_VEL
LIN {X 0,Y 271.321,Z 259.267,A -85,B 0,C 180,E1 -17685.623,E2 -17685.623} C_VEL
LIN {X 0,Y 271.575,Z 263.074,A -85,B 0,C 180,E1 -17689.686,E2 -17689.686} C_VEL
LIN {X 0,Y 271.51,Z 264.985,A -85,B 0,C 180,E1 -17691.593,E2 -17691.593} C_VEL
LIN {X 0,Y 270.936,Z 268.801,A -85,B 0,C 180,E1 -17695.203,E2 -17695.203} C_VEL
LIN {X 0,Y 270.736,Z 270.284,A -85,B 0,C 180,E1 -17696.551,E2 -17696.551} C_VEL
LIN {X 0,Y 271.736,Z 273.571,A -85,B 0,C 180,E1 -17696.81,E2 -17696.81} C_VEL
LIN {X 0,Y 275.98,Z 285.719,A -85,B 0,C 180,E1 -17697.974,E2 -17697.974} C_VEL
LIN {X 0,Y 279.282,Z 297.858,A -85,B 0,C 180,E1 -17699.22,E2 -17699.22} C_VEL
LIN {X 0,Y 281.885,Z 311.577,A -85,B 0,C 180,E1 -17700.765,E2 -17700.765} C_VEL
LIN {X 0,Y 283.32,Z 323.538,A -85,B 0,C 180,E1 -17702.282,E2 -17702.282} C_VEL
LIN {X 0,Y 283.609,Z 328.167,A -85,B 0,C 180,E1 -17702.913,E2 -17702.913} C_VEL
LIN {X 0,Y 281.689,Z 338.66,A -85,B 0,C 180,E1 -17704.272,E2 -17704.272} C_VEL
LIN {X 0,Y 279.384,Z 348.954,A -85,B 0,C 180,E1 -17705.872,E2 -17705.872} C_VEL
LIN {X 0,Y 277.082,Z 358.341,A -85,B 0,C 180,E1 -17707.637,E2 -17707.637} C_VEL
LIN {X 0,Y 274.804,Z 367.791,A -85,B 0,C 180,E1 -17709.802,E2 -17709.802} C_VEL
LIN {X 0,Y 272.924,Z 375.625,A -85,B 0,C 180,E1 -17712,E2 -17712} C_VEL
LIN {X 0,Y 271.396,Z 382.146,A -85,B 0,C 180,E1 -17714.222,E2 -17714.222} C_VEL
LIN {X 0,Y 270.144,Z 387.56,A -85,B 0,C 180,E1 -17716.459,E2 -17716.459} C_VEL
LIN {X 0,Y 268.989,Z 393.26,A -85,B 0,C 180,E1 -17719.462,E2 -17719.462} C_VEL
LIN {X 0,Y 268.369,Z 397.399,A -85,B 0,C 180,E1 -17722.476,E2 -17722.476} C_VEL
LIN {X 0,Y 268.131,Z 400.104,A -85,B 0,C 180,E1 -17725.49,E2 -17725.49} C_VEL
LIN {X 0,Y 268.13,Z 401.442,A -85,B 0,C 180,E1 -17728.498,E2 -17728.498} C_VEL
LIN {X 0,Y 268.155,Z 401.607,A -85,B 0,C 180,E1 -17730,E2 -17730} C_VEL
LIN {X 0,Y 268.106,Z 400.929,A -85,B 0,C 180,E1 -17733.005,E2 -17733.005} C_VEL
LIN {X 0,Y 268.22,Z 398.902,A -85,B 0,C 180,E1 -17736.016,E2 -17736.016} C_VEL
LIN {X 0,Y 268.649,Z 395.479,A -85,B 0,C 180,E1 -17739.031,E2 -17739.031} C_VEL
LIN {X 0,Y 269.436,Z 390.558,A -85,B 0,C 180,E1 -17742.044,E2 -17742.044} C_VEL
LIN {X 0,Y 270.952,Z 384.002,A -85,B 0,C 180,E1 -17745.033,E2 -17745.033} C_VEL
LIN {X 0,Y 272.493,Z 377.113,A -85,B 0,C 180,E1 -17747.5,E2 -17747.5} C_VEL
LIN {X 0,Y 274.436,Z 369.065,A -85,B 0,C 180,E1 -17749.835,E2 -17749.835} C_VEL
LIN {X 0,Y 276.693,Z 359.9,A -85,B 0,C 180,E1 -17752.003,E2 -17752.003} C_VEL
LIN {X 0,Y 278.847,Z 350.765,A -85,B 0,C 180,E1 -17753.782,E2 -17753.782} C_VEL
LIN {X 0,Y 281.491,Z 339.211,A -85,B 0,C 180,E1 -17755.622,E2 -17755.622} C_VEL
LIN {X 0,Y 283.579,Z 327.94,A -85,B 0,C 180,E1 -17757.09,E2 -17757.09} C_VEL
LIN {X 0,Y 282.378,Z 314.799,A -85,B 0,C 180,E1 -17758.814,E2 -17758.814} C_VEL
LIN {X 0,Y 280.142,Z 301.97,A -85,B 0,C 180,E1 -17760.31,E2 -17760.31} C_VEL
LIN {X 0,Y 277.037,Z 289.296,A -85,B 0,C 180,E1 -17761.639,E2 -17761.639} C_VEL
LIN {X 0,Y 272.568,Z 275.764,A -85,B 0,C 180,E1 -17762.951,E2 -17762.951} C_VEL
LIN {X 0,Y 270.776,Z 270.932,A -85,B 0,C 180,E1 -17763.378,E2 -17763.378} C_VEL
LIN {X 0,Y 270.7,Z 270.155,A -85,B 0,C 180,E1 -17763.485,E2 -17763.485} C_VEL
LIN {X 0,Y 271.238,Z 266.854,A -85,B 0,C 180,E1 -17766.58,E2 -17766.58} C_VEL
LIN {X 0,Y 271.558,Z 264.266,A -85,B 0,C 180,E1 -17769.067,E2 -17769.067} C_VEL
LIN {X 0,Y 271.447,Z 261.128,A -85,B 0,C 180,E1 -17772.312,E2 -17772.312} C_VEL
LIN {X 0,Y 271.082,Z 258.17,A -85,B 0,C 180,E1 -17775.573,E2 -17775.573} C_VEL
LIN {X 0,Y 270.621,Z 254.816,A -85,B 0,C 180,E1 -17779.515,E2 -17779.515} C_VEL
LIN {X 0,Y 270.272,Z 252.582,A -85,B 0,C 180,E1 -17782.332,E2 -17782.332} C_VEL
LIN {X 0,Y 270.202,Z 252.456,A -85,B 0,C 180,E1 -17786.892,E2 -17786.892} C_VEL
LIN {X 0,Y 270.183,Z 252.456,A -85,B 0,C 180,E1 -17790.381,E2 -17790.381} C_VEL
LIN {X 0,Y 270.203,Z 252.454,A -85,B 0,C 180,E1 -17793.758,E2 -17793.758} C_VEL
LIN {X 0,Y 270.203,Z 252.454,A -85,B 0,C 180,E1 -17797.036,E2 -17797.036} C_VEL
LIN {X 0,Y 270.264,Z 252.445,A -85,B 0,C 180,E1 -17800.242,E2 -17800.242} C_VEL
LIN {X 0,Y 270.374,Z 252.429,A -85,B 0,C 180,E1 -17804.934,E2 -17804.934} C_VEL
LIN {X 0,Y 270.411,Z 252.419,A -85,B 0,C 180,E1 -17809.518,E2 -17809.518} C_VEL
LIN {X 0,Y 270.564,Z 252.406,A -85,B 0,C 180,E1 -17812.538,E2 -17812.538} C_VEL
LIN {X 0,Y 270.787,Z 252.38,A -85,B 0,C 180,E1 -17818.513,E2 -17818.513} C_VEL
LIN {X 0,Y 270.784,Z 252.38,A -85,B 0,C 180,E1 -17821.487,E2 -17821.487} C_VEL
LIN {X 0,Y 270.6,Z 252.402,A -85,B 0,C 180,E1 -17827.462,E2 -17827.462} C_VEL
LIN {X 0,Y 270.415,Z 252.426,A -85,B 0,C 180,E1 -17830.482,E2 -17830.482} C_VEL
LIN {X 0,Y 270.405,Z 252.428,A -85,B 0,C 180,E1 -17835.065,E2 -17835.065} C_VEL
LIN {X 0,Y 270.303,Z 252.439,A -85,B 0,C 180,E1 -17839.756,E2 -17839.756} C_VEL
LIN {X 0,Y 270.239,Z 252.449,A -85,B 0,C 180,E1 -17844.589,E2 -17844.589} C_VEL
LIN {X 0,Y 270.271,Z 252.443,A -85,B 0,C 180,E1 -17847.909,E2 -17847.909} C_VEL
LIN {X 0,Y 270.185,Z 252.455,A -85,B 0,C 180,E1 -17851.348,E2 -17851.348} C_VEL
LIN {X 0,Y 270.199,Z 252.454,A -85,B 0,C 180,E1 -17854.906,E2 -17854.906} C_VEL
LIN {X 0,Y 270.198,Z 252.455,A -85,B 0,C 180,E1 -17858.711,E2 -17858.711} C_VEL
LIN {X 0,Y 270.158,Z 252.46,A -85,B 0,C 180,E1 -17863.247,E2 -17863.247} C_VEL
LIN {X 0,Y 270.225,Z 252.787,A -85,B 0,C 180,E1 -17864.605,E2 -17864.605} C_VEL
LIN {X 0,Y 270.616,Z 255.881,A -85,B 0,C 180,E1 -17868.864,E2 -17868.864} C_VEL
LIN {X 0,Y 270.627,Z 257.916,A -85,B 0,C 180,E1 -17871.445,E2 -17871.445} C_VEL
LIN {X 0,Y 270.346,Z 260.948,A -85,B 0,C 180,E1 -17875.116,E2 -17875.116} C_VEL
LIN {X 0,Y 270.216,Z 262.215,A -85,B 0,C 180,E1 -17876.577,E2 -17876.577} C_VEL
LIN {X 0,Y 271.297,Z 265.469,A -85,B 0,C 180,E1 -17876.855,E2 -17876.855} C_VEL
LIN {X 0,Y 276.304,Z 278.301,A -85,B 0,C 180,E1 -17878.187,E2 -17878.187} C_VEL
LIN {X 0,Y 280.291,Z 291.238,A -85,B 0,C 180,E1 -17879.627,E2 -17879.627} C_VEL
LIN {X 0,Y 283.244,Z 304.445,A -85,B 0,C 180,E1 -17881.228,E2 -17881.228} C_VEL
LIN {X 0,Y 284.834,Z 315.062,A -85,B 0,C 180,E1 -17882.656,E2 -17882.656} C_VEL
LIN {X 0,Y 282.676,Z 327.505,A -85,B 0,C 180,E1 -17884.209,E2 -17884.209} C_VEL
LIN {X 0,Y 280.211,Z 338.851,A -85,B 0,C 180,E1 -17885.948,E2 -17885.948} C_VEL
LIN {X 0,Y 278.047,Z 348.251,A -85,B 0,C 180,E1 -17887.719,E2 -17887.719} C_VEL
LIN {X 0,Y 275.647,Z 357.698,A -85,B 0,C 180,E1 -17889.867,E2 -17889.867} C_VEL
LIN {X 0,Y 273.355,Z 366.703,A -85,B 0,C 180,E1 -17892.417,E2 -17892.417} C_VEL
LIN {X 0,Y 272.163,Z 372.023,A -85,B 0,C 180,E1 -17894.268,E2 -17894.268} C_VEL
LIN {X 0,Y 270.703,Z 377.424,A -85,B 0,C 180,E1 -17896.488,E2 -17896.488} C_VEL
LIN {X 0,Y 269.498,Z 383.094,A -85,B 0,C 180,E1 -17899.482,E2 -17899.482} C_VEL
LIN {X 0,Y 268.727,Z 387.212,A -85,B 0,C 180,E1 -17902.486,E2 -17902.486} C_VEL
LIN {X 0,Y 268.314,Z 389.904,A -85,B 0,C 180,E1 -17905.493,E2 -17905.493} C_VEL
LIN {X 0,Y 268.182,Z 391.249,A -85,B 0,C 180,E1 -17908.498,E2 -17908.498} C_VEL
LIN {X 0,Y 268.182,Z 391.278,A -85,B 0,C 180,E1 -17911.502,E2 -17911.502} C_VEL
LIN {X 0,Y 268.311,Z 389.988,A -85,B 0,C 180,E1 -17914.507,E2 -17914.507} C_VEL
LIN {X 0,Y 268.727,Z 387.348,A -85,B 0,C 180,E1 -17917.514,E2 -17917.514} C_VEL
LIN {X 0,Y 269.48,Z 383.287,A -85,B 0,C 180,E1 -17920.519,E2 -17920.519} C_VEL
LIN {X 0,Y 270.653,Z 377.677,A -85,B 0,C 180,E1 -17923.515,E2 -17923.515} C_VEL
LIN {X 0,Y 272.41,Z 371.333,A -85,B 0,C 180,E1 -17926.102,E2 -17926.102} C_VEL
LIN {X 0,Y 274.077,Z 363.698,A -85,B 0,C 180,E1 -17928.618,E2 -17928.618} C_VEL
LIN {X 0,Y 276.302,Z 355.199,A -85,B 0,C 180,E1 -17930.861,E2 -17930.861} C_VEL
LIN {X 0,Y 278.765,Z 345.251,A -85,B 0,C 180,E1 -17933.003,E2 -17933.003} C_VEL
LIN {X 0,Y 281.332,Z 334.173,A -85,B 0,C 180,E1 -17934.933,E2 -17934.933} C_VEL
LIN {X 0,Y 283.643,Z 323.139,A -85,B 0,C 180,E1 -17936.487,E2 -17936.487} C_VEL
LIN {X 0,Y 284.899,Z 315.437,A -85,B 0,C 180,E1 -17937.412,E2 -17937.412} C_VEL
LIN {X 0,Y 283.176,Z 303.784,A -85,B 0,C 180,E1 -17938.972,E2 -17938.972} C_VEL
LIN {X 0,Y 280.355,Z 291.29,A -85,B 0,C 180,E1 -17940.488,E2 -17940.488} C_VEL
LIN {X 0,Y 276.388,Z 278.489,A -85,B 0,C 180,E1 -17941.921,E2 -17941.921} C_VEL
LIN {X 0,Y 271.497,Z 265.778,A -85,B 0,C 180,E1 -17943.237,E2 -17943.237} C_VEL
LIN {X 0,Y 270.343,Z 262.984,A -85,B 0,C 180,E1 -17943.502,E2 -17943.502} C_VEL
LIN {X 0,Y 270.229,Z 262.172,A -85,B 0,C 180,E1 -17943.606,E2 -17943.606} C_VEL
LIN {X 0,Y 270.51,Z 259.54,A -85,B 0,C 180,E1 -17946.695,E2 -17946.695} C_VEL
LIN {X 0,Y 270.64,Z 257.812,A -85,B 0,C 180,E1 -17948.827,E2 -17948.827} C_VEL
LIN {X 0,Y 270.614,Z 255.994,A -85,B 0,C 180,E1 -17951.136,E2 -17951.136} C_VEL
LIN {X 0,Y 270.289,Z 253.457,A -85,B 0,C 180,E1 -17954.592,E2 -17954.592} C_VEL
LIN {X 0,Y 270.159,Z 252.462,A -85,B 0,C 180,E1 -17956.753,E2 -17956.753} C_VEL
LIN {X 0,Y 270.209,Z 252.454,A -85,B 0,C 180,E1 -17961.374,E2 -17961.374} C_VEL
LIN {X 0,Y 270.2,Z 252.453,A -85,B 0,C 180,E1 -17965.094,E2 -17965.094} C_VEL
LIN {X 0,Y 270.203,Z 252.454,A -85,B 0,C 180,E1 -17969.131,E2 -17969.131} C_VEL
LIN {X 0,Y 270.267,Z 252.446,A -85,B 0,C 180,E1 -17972.146,E2 -17972.146} C_VEL
LIN {X 0,Y 270.24,Z 252.443,A -85,B 0,C 180,E1 -17975.538,E2 -17975.538} C_VEL
LIN {X 0,Y 270.304,Z 252.439,A -85,B 0,C 180,E1 -17980.244,E2 -17980.244} C_VEL
LIN {X 0,Y 270.406,Z 252.426,A -85,B 0,C 180,E1 -17984.935,E2 -17984.935} C_VEL
LIN {X 0,Y 270.413,Z 252.424,A -85,B 0,C 180,E1 -17989.518,E2 -17989.518} C_VEL
LIN {X 0,Y 270.587,Z 252.404,A -85,B 0,C 180,E1 -17992.538,E2 -17992.538} C_VEL
LIN {X 0,Y 270.781,Z 252.383,A -85,B 0,C 180,E1 -17998.513,E2 -17998.513} C_VEL
LIN {X 0,Y 270.789,Z 252.381,A -85,B 0,C 180,E1 -18001.487,E2 -18001.487} C_VEL
LIN {X 0,Y 270.565,Z 252.405,A -85,B 0,C 180,E1 -18007.462,E2 -18007.462} C_VEL
LIN {X 0,Y 270.529,Z 252.412,A -85,B 0,C 180,E1 -18008.952,E2 -18008.952} C_VEL
LIN {X 0,Y 269.893,Z 252.499,A -85,B 0,C 180,E1 -18010.192,E2 -18010.192} C_VEL
LIN {X 0,Y 267.015,Z 252.86,A -85,B 0,C 180,E1 -18012.211,E2 -18012.211} C_VEL
LIN {X 0,Y 264.523,Z 253.165,A -85,B 0,C 180,E1 -18013.853,E2 -18013.853} C_VEL
LIN {X 0,Y 263.419,Z 253.299,A -85,B 0,C 180,E1 -18015.127,E2 -18015.127} C_VEL
LIN {X 0,Y 263.312,Z 253.312,A -85,B 0,C 180,E1 -18015.559,E2 -18015.559} C_VEL
LIN {X 0,Y 263.246,Z 253.32,A -85,B 0,C 180,E1 -18020.308,E2 -18020.308} C_VEL
LIN {X 0,Y 263.169,Z 253.322,A -85,B 0,C 180,E1 -18025.295,E2 -18025.295} C_VEL
LIN {X 0,Y 263.135,Z 253.333,A -85,B 0,C 180,E1 -18028.735,E2 -18028.735} C_VEL
LIN {X 0,Y 263.13,Z 253.335,A -85,B 0,C 180,E1 -18032.289,E2 -18032.289} C_VEL
LIN {X 0,Y 263.199,Z 253.394,A -85,B 0,C 180,E1 -18036.849,E2 -18036.849} C_VEL
LIN {X 0,Y 263.552,Z 255.622,A -85,B 0,C 180,E1 -18039.791,E2 -18039.791} C_VEL
LIN {X 0,Y 264.094,Z 259.107,A -85,B 0,C 180,E1 -18044.067,E2 -18044.067} C_VEL
LIN {X 0,Y 264.375,Z 261.03,A -85,B 0,C 180,E1 -18046.277,E2 -18046.277} C_VEL
LIN {X 0,Y 264.512,Z 262.941,A -85,B 0,C 180,E1 -18048.375,E2 -18048.375} C_VEL
LIN {X 0,Y 264.556,Z 264.838,A -85,B 0,C 180,E1 -18050.389,E2 -18050.389} C_VEL
LIN {X 0,Y 264.04,Z 268.642,A -85,B 0,C 180,E1 -18054.156,E2 -18054.156} C_VEL
LIN {X 0,Y 263.846,Z 270.086,A -85,B 0,C 180,E1 -18055.542,E2 -18055.542} C_VEL
LIN {X 0,Y 264.779,Z 273.286,A -85,B 0,C 180,E1 -18055.814,E2 -18055.814} C_VEL
LIN {X 0,Y 268.889,Z 284.491,A -85,B 0,C 180,E1 -18056.958,E2 -18056.958} C_VEL
LIN {X 0,Y 272.506,Z 297.255,A -85,B 0,C 180,E1 -18058.329,E2 -18058.329} C_VEL
LIN {X 0,Y 275.115,Z 310.708,A -85,B 0,C 180,E1 -18059.896,E2 -18059.896} C_VEL
LIN {X 0,Y 276.685,Z 323.4,A -85,B 0,C 180,E1 -18061.558,E2 -18061.558} C_VEL
LIN {X 0,Y 277.046,Z 329.466,A -85,B 0,C 180,E1 -18062.422,E2 -18062.422} C_VEL
LIN {X 0,Y 274.818,Z 340.611,A -85,B 0,C 180,E1 -18063.941,E2 -18063.941} C_VEL
LIN {X 0,Y 272.361,Z 350.789,A -85,B 0,C 180,E1 -18065.615,E2 -18065.615} C_VEL
LIN {X 0,Y 269.675,Z 361.527,A -85,B 0,C 180,E1 -18067.797,E2 -18067.797} C_VEL
LIN {X 0,Y 267.361,Z 370.396,A -85,B 0,C 180,E1 -18070.018,E2 -18070.018} C_VEL
LIN {X 0,Y 265.462,Z 378.078,A -85,B 0,C 180,E1 -18072.38,E2 -18072.38} C_VEL
LIN {X 0,Y 264.044,Z 383.938,A -85,B 0,C 180,E1 -18074.563,E2 -18074.563} C_VEL
LIN {X 0,Y 262.81,Z 389.041,A -85,B 0,C 180,E1 -18076.861,E2 -18076.861} C_VEL
LIN {X 0,Y 261.757,Z 394.31,A -85,B 0,C 180,E1 -18079.949,E2 -18079.949} C_VEL
LIN {X 0,Y 261.31,Z 397.265,A -85,B 0,C 180,E1 -18082.271,E2 -18082.271} C_VEL
LIN {X 0,Y 261.046,Z 399.969,A -85,B 0,C 180,E1 -18085.367,E2 -18085.367} C_VEL
LIN {X 0,Y 261.037,Z 401.308,A -85,B 0,C 180,E1 -18088.457,E2 -18088.457} C_VEL
LIN {X 0,Y 261.082,Z 401.473,A -85,B 0,C 180,E1 -18090,E2 -18090} C_VEL
LIN {X 0,Y 261.005,Z 400.794,A -85,B 0,C 180,E1 -18093.087,E2 -18093.087} C_VEL
LIN {X 0,Y 261.145,Z 398.767,A -85,B 0,C 180,E1 -18096.18,E2 -18096.18} C_VEL
LIN {X 0,Y 261.588,Z 395.343,A -85,B 0,C 180,E1 -18099.276,E2 -18099.276} C_VEL
LIN {X 0,Y 262.448,Z 390.422,A -85,B 0,C 180,E1 -18102.37,E2 -18102.37} C_VEL
LIN {X 0,Y 263.632,Z 385.683,A -85,B 0,C 180,E1 -18104.67,E2 -18104.67} C_VEL
LIN {X 0,Y 265.076,Z 379.908,A -85,B 0,C 180,E1 -18106.956,E2 -18106.956} C_VEL
LIN {X 0,Y 267.029,Z 371.645,A -85,B 0,C 180,E1 -18109.607,E2 -18109.607} C_VEL
LIN {X 0,Y 269.228,Z 363.025,A -85,B 0,C 180,E1 -18111.838,E2 -18111.838} C_VEL
LIN {X 0,Y 271.848,Z 352.582,A -85,B 0,C 180,E1 -18114.028,E2 -18114.028} C_VEL
LIN {X 0,Y 274.398,Z 342.084,A -85,B 0,C 180,E1 -18115.811,E2 -18115.811} C_VEL
LIN {X 0,Y 276.817,Z 330.659,A -85,B 0,C 180,E1 -18117.398,E2 -18117.398} C_VEL
LIN {X 0,Y 276.835,Z 326.319,A -85,B 0,C 180,E1 -18118.012,E2 -18118.012} C_VEL
LIN {X 0,Y 275.697,Z 314.519,A -85,B 0,C 180,E1 -18119.595,E2 -18119.595} C_VEL
LIN {X 0,Y 273.285,Z 300.891,A -85,B 0,C 180,E1 -18121.231,E2 -18121.231} C_VEL
LIN {X 0,Y 270.065,Z 288.414,A -85,B 0,C 180,E1 -18122.603,E2 -18122.603} C_VEL
LIN {X 0,Y 266.048,Z 276.615,A -85,B 0,C 180,E1 -18123.816,E2 -18123.816} C_VEL
LIN {X 0,Y 263.911,Z 270.966,A -85,B 0,C 180,E1 -18124.357,E2 -18124.357} C_VEL
LIN {X 0,Y 263.808,Z 270.08,A -85,B 0,C 180,E1 -18124.427,E2 -18124.427} C_VEL
LIN {X 0,Y 264.332,Z 266.689,A -85,B 0,C 180,E1 -18127.699,E2 -18127.699} C_VEL
LIN {X 0,Y 264.536,Z 264.792,A -85,B 0,C 180,E1 -18129.614,E2 -18129.614} C_VEL
LIN {X 0,Y 264.48,Z 262.621,A -85,B 0,C 180,E1 -18131.923,E2 -18131.923} C_VEL
LIN {X 0,Y 264.299,Z 260.638,A -85,B 0,C 180,E1 -18134.114,E2 -18134.114} C_VEL
LIN {X 0,Y 263.807,Z 257.142,A -85,B 0,C 180,E1 -18138.24,E2 -18138.24} C_VEL
LIN {X 0,Y 263.198,Z 253.411,A -85,B 0,C 180,E1 -18143.058,E2 -18143.058} C_VEL
LIN {X 0,Y 263.151,Z 253.335,A -85,B 0,C 180,E1 -18145.886,E2 -18145.886} C_VEL
LIN {X 0,Y 263.126,Z 253.336,A -85,B 0,C 180,E1 -18149.504,E2 -18149.504} C_VEL
LIN {X 0,Y 263.142,Z 253.332,A -85,B 0,C 180,E1 -18152.997,E2 -18152.997} C_VEL
LIN {X 0,Y 263.147,Z 253.332,A -85,B 0,C 180,E1 -18156.384,E2 -18156.384} C_VEL
LIN {X 0,Y 263.24,Z 253.32,A -85,B 0,C 180,E1 -18159.692,E2 -18159.692} C_VEL
LIN {X 0,Y 263.316,Z 253.31,A -85,B 0,C 180,E1 -18164.52,E2 -18164.52} C_VEL
LIN {X 0,Y 263.354,Z 253.298,A -85,B 0,C 180,E1 -18169.234,E2 -18169.234} C_VEL
LIN {X 0,Y 263.528,Z 253.283,A -85,B 0,C 180,E1 -18172.337,E2 -18172.337} C_VEL
LIN {X 0,Y 263.752,Z 253.257,A -85,B 0,C 180,E1 -18178.473,E2 -18178.473} C_VEL
LIN {X 0,Y 263.749,Z 253.256,A -85,B 0,C 180,E1 -18181.527,E2 -18181.527} C_VEL
LIN {X 0,Y 263.56,Z 253.28,A -85,B 0,C 180,E1 -18187.662,E2 -18187.662} C_VEL
LIN {X 0,Y 263.357,Z 253.306,A -85,B 0,C 180,E1 -18190.766,E2 -18190.766} C_VEL
LIN {X 0,Y 263.353,Z 253.305,A -85,B 0,C 180,E1 -18195.478,E2 -18195.478} C_VEL
LIN {X 0,Y 263.264,Z 253.315,A -85,B 0,C 180,E1 -18200.307,E2 -18200.307} C_VEL
LIN {X 0,Y 263.194,Z 253.325,A -85,B 0,C 180,E1 -18205.293,E2 -18205.293} C_VEL
LIN {X 0,Y 263.167,Z 253.329,A -85,B 0,C 180,E1 -18208.731,E2 -18208.731} C_VEL
LIN {X 0,Y 263.134,Z 253.334,A -85,B 0,C 180,E1 -18212.288,E2 -18212.288} C_VEL
LIN {X 0,Y 263.177,Z 253.328,A -85,B 0,C 180,E1 -18216.761,E2 -18216.761} C_VEL
LIN {X 0,Y 263.092,Z 253.337,A -85,B 0,C 180,E1 -18219.875,E2 -18219.875} C_VEL
LIN {X 0,Y 263.137,Z 253.498,A -85,B 0,C 180,E1 -18223.852,E2 -18223.852} C_VEL
LIN {X 0,Y 263.543,Z 256.54,A -85,B 0,C 180,E1 -18228.188,E2 -18228.188} C_VEL
LIN {X 0,Y 263.612,Z 258.374,A -85,B 0,C 180,E1 -18230.638,E2 -18230.638} C_VEL
LIN {X 0,Y 263.415,Z 261.106,A -85,B 0,C 180,E1 -18234.058,E2 -18234.058} C_VEL
LIN {X 0,Y 263.261,Z 262.386,A -85,B 0,C 180,E1 -18235.579,E2 -18235.579} C_VEL
LIN {X 0,Y 264.341,Z 265.571,A -85,B 0,C 180,E1 -18235.862,E2 -18235.862} C_VEL
LIN {X 0,Y 268.204,Z 274.982,A -85,B 0,C 180,E1 -18236.891,E2 -18236.891} C_VEL
LIN {X 0,Y 271.87,Z 285.716,A -85,B 0,C 180,E1 -18238.112,E2 -18238.112} C_VEL
LIN {X 0,Y 275.099,Z 297.649,A -85,B 0,C 180,E1 -18239.567,E2 -18239.567} C_VEL
LIN {X 0,Y 277.534,Z 310.267,A -85,B 0,C 180,E1 -18241.24,E2 -18241.24} C_VEL
LIN {X 0,Y 278.309,Z 316.359,A -85,B 0,C 180,E1 -18242.109,E2 -18242.109} C_VEL
LIN {X 0,Y 276.307,Z 327.644,A -85,B 0,C 180,E1 -18243.569,E2 -18243.569} C_VEL
LIN {X 0,Y 273.745,Z 338.989,A -85,B 0,C 180,E1 -18245.342,E2 -18245.342} C_VEL
LIN {X 0,Y 271.467,Z 348.39,A -85,B 0,C 180,E1 -18247.149,E2 -18247.149} C_VEL
LIN {X 0,Y 268.964,Z 357.836,A -85,B 0,C 180,E1 -18249.344,E2 -18249.344} C_VEL
LIN {X 0,Y 266.546,Z 366.864,A -85,B 0,C 180,E1 -18251.961,E2 -18251.961} C_VEL
LIN {X 0,Y 265.324,Z 372.16,A -85,B 0,C 180,E1 -18253.852,E2 -18253.852} C_VEL
LIN {X 0,Y 263.773,Z 377.56,A -85,B 0,C 180,E1 -18256.126,E2 -18256.126} C_VEL
LIN {X 0,Y 262.511,Z 383.23,A -85,B 0,C 180,E1 -18259.199,E2 -18259.199} C_VEL
LIN {X 0,Y 261.673,Z 387.348,A -85,B 0,C 180,E1 -18262.283,E2 -18262.283} C_VEL
LIN {X 0,Y 261.234,Z 390.039,A -85,B 0,C 180,E1 -18265.371,E2 -18265.371} C_VEL
LIN {X 0,Y 261.09,Z 391.384,A -85,B 0,C 180,E1 -18268.458,E2 -18268.458} C_VEL
LIN {X 0,Y 261.09,Z 391.413,A -85,B 0,C 180,E1 -18271.543,E2 -18271.543} C_VEL
LIN {X 0,Y 261.23,Z 390.123,A -85,B 0,C 180,E1 -18274.63,E2 -18274.63} C_VEL
LIN {X 0,Y 261.672,Z 387.482,A -85,B 0,C 180,E1 -18277.718,E2 -18277.718} C_VEL
LIN {X 0,Y 262.476,Z 383.422,A -85,B 0,C 180,E1 -18280.803,E2 -18280.803} C_VEL
LIN {X 0,Y 263.726,Z 377.811,A -85,B 0,C 180,E1 -18283.877,E2 -18283.877} C_VEL
LIN {X 0,Y 265.579,Z 371.467,A -85,B 0,C 180,E1 -18286.528,E2 -18286.528} C_VEL
LIN {X 0,Y 267.037,Z 364.936,A -85,B 0,C 180,E1 -18288.768,E2 -18288.768} C_VEL
LIN {X 0,Y 269.254,Z 356.812,A -85,B 0,C 180,E1 -18291.033,E2 -18291.033} C_VEL
LIN {X 0,Y 271.783,Z 347.159,A -85,B 0,C 180,E1 -18293.226,E2 -18293.226} C_VEL
LIN {X 0,Y 274.407,Z 336.443,A -85,B 0,C 180,E1 -18295.201,E2 -18295.201} C_VEL
LIN {X 0,Y 277.02,Z 324.565,A -85,B 0,C 180,E1 -18296.968,E2 -18296.968} C_VEL
LIN {X 0,Y 278.391,Z 317.003,A -85,B 0,C 180,E1 -18297.922,E2 -18297.922} C_VEL
LIN {X 0,Y 276.748,Z 305.28,A -85,B 0,C 180,E1 -18299.567,E2 -18299.567} C_VEL
LIN {X 0,Y 273.756,Z 291.909,A -85,B 0,C 180,E1 -18301.265,E2 -18301.265} C_VEL
LIN {X 0,Y 269.654,Z 278.888,A -85,B 0,C 180,E1 -18302.801,E2 -18302.801} C_VEL
LIN {X 0,Y 265.737,Z 268.771,A -85,B 0,C 180,E1 -18303.922,E2 -18303.922} C_VEL
LIN {X 0,Y 263.403,Z 263.168,A -85,B 0,C 180,E1 -18304.505,E2 -18304.505} C_VEL
LIN {X 0,Y 263.291,Z 262.342,A -85,B 0,C 180,E1 -18304.578,E2 -18304.578} C_VEL
LIN {X 0,Y 263.526,Z 259.7,A -85,B 0,C 180,E1 -18307.835,E2 -18307.835} C_VEL
LIN {X 0,Y 263.605,Z 258.162,A -85,B 0,C 180,E1 -18309.782,E2 -18309.782} C_VEL
LIN {X 0,Y 263.544,Z 256.633,A -85,B 0,C 180,E1 -18311.812,E2 -18311.812} C_VEL
LIN {X 0,Y 263.138,Z 253.608,A -85,B 0,C 180,E1 -18316.148,E2 -18316.148} C_VEL
LIN {X 0,Y 263.111,Z 253.338,A -85,B 0,C 180,E1 -18318.41,E2 -18318.41} C_VEL
LIN {X 0,Y 263.159,Z 253.33,A -85,B 0,C 180,E1 -18322.103,E2 -18322.103} C_VEL
LIN {X 0,Y 263.153,Z 253.332,A -85,B 0,C 180,E1 -18325.886,E2 -18325.886} C_VEL
LIN {X 0,Y 263.153,Z 253.332,A -85,B 0,C 180,E1 -18329.507,E2 -18329.507} C_VEL
LIN {X 0,Y 263.194,Z 253.326,A -85,B 0,C 180,E1 -18333.003,E2 -18333.003} C_VEL
LIN {X 0,Y 263.158,Z 253.33,A -85,B 0,C 180,E1 -18336.384,E2 -18336.384} C_VEL
LIN {X 0,Y 263.266,Z 253.315,A -85,B 0,C 180,E1 -18339.693,E2 -18339.693} C_VEL
LIN {X 0,Y 263.354,Z 253.304,A -85,B 0,C 180,E1 -18344.522,E2 -18344.522} C_VEL
LIN {X 0,Y 263.356,Z 253.303,A -85,B 0,C 180,E1 -18349.233,E2 -18349.233} C_VEL
LIN {X 0,Y 263.547,Z 253.281,A -85,B 0,C 180,E1 -18352.338,E2 -18352.338} C_VEL
LIN {X 0,Y 263.746,Z 253.259,A -85,B 0,C 180,E1 -18358.473,E2 -18358.473} C_VEL
LIN {X 0,Y 263.753,Z 253.258,A -85,B 0,C 180,E1 -18361.527,E2 -18361.527} C_VEL
LIN {X 0,Y 263.529,Z 253.282,A -85,B 0,C 180,E1 -18367.663,E2 -18367.663} C_VEL
LIN {X 0,Y 263.352,Z 253.307,A -85,B 0,C 180,E1 -18370.766,E2 -18370.766} C_VEL
LIN {X 0,Y 263.312,Z 253.312,A -85,B 0,C 180,E1 -18375.559,E2 -18375.559} C_VEL
LIN {X 0,Y 262.583,Z 253.403,A -85,B 0,C 180,E1 -18376.835,E2 -18376.835} C_VEL
LIN {X 0,Y 259.659,Z 253.765,A -85,B 0,C 180,E1 -18378.911,E2 -18378.911} C_VEL
LIN {X 0,Y 257.208,Z 254.072,A -85,B 0,C 180,E1 -18380.6,E2 -18380.6} C_VEL
LIN {X 0,Y 256.162,Z 254.202,A -85,B 0,C 180,E1 -18381.911,E2 -18381.911} C_VEL
LIN {X 0,Y 256.079,Z 254.211,A -85,B 0,C 180,E1 -18382.356,E2 -18382.356} C_VEL
LIN {X 0,Y 256.1,Z 254.203,A -85,B 0,C 180,E1 -18386.045,E2 -18386.045} C_VEL
LIN {X 0,Y 256.056,Z 254.215,A -85,B 0,C 180,E1 -18389.607,E2 -18389.607} C_VEL
LIN {X 0,Y 256.067,Z 254.213,A -85,B 0,C 180,E1 -18393.293,E2 -18393.293} C_VEL
LIN {X 0,Y 256.084,Z 254.216,A -85,B 0,C 180,E1 -18395.193,E2 -18395.193} C_VEL
LIN {X 0,Y 256.32,Z 255.106,A -85,B 0,C 180,E1 -18397.33,E2 -18397.33} C_VEL
LIN {X 0,Y 256.715,Z 257.928,A -85,B 0,C 180,E1 -18401.075,E2 -18401.075} C_VEL
LIN {X 0,Y 257.238,Z 261.323,A -85,B 0,C 180,E1 -18405.263,E2 -18405.263} C_VEL
LIN {X 0,Y 257.498,Z 264.704,A -85,B 0,C 180,E1 -18409.077,E2 -18409.077} C_VEL
LIN {X 0,Y 257.313,Z 267.827,A -85,B 0,C 180,E1 -18412.38,E2 -18412.38} C_VEL
LIN {X 0,Y 256.968,Z 270.047,A -85,B 0,C 180,E1 -18414.5,E2 -18414.5} C_VEL
LIN {X 0,Y 258.027,Z 273.355,A -85,B 0,C 180,E1 -18414.798,E2 -18414.798} C_VEL
LIN {X 0,Y 262.464,Z 285.418,A -85,B 0,C 180,E1 -18416.108,E2 -18416.108} C_VEL
LIN {X 0,Y 266.233,Z 298.88,A -85,B 0,C 180,E1 -18417.643,E2 -18417.643} C_VEL
LIN {X 0,Y 268.649,Z 311.719,A -85,B 0,C 180,E1 -18419.219,E2 -18419.219} C_VEL
LIN {X 0,Y 270.081,Z 323.262,A -85,B 0,C 180,E1 -18420.796,E2 -18420.796} C_VEL
LIN {X 0,Y 270.467,Z 330.763,A -85,B 0,C 180,E1 -18421.902,E2 -18421.902} C_VEL
LIN {X 0,Y 268.014,Z 342.148,A -85,B 0,C 180,E1 -18423.526,E2 -18423.526} C_VEL
LIN {X 0,Y 265.373,Z 352.612,A -85,B 0,C 180,E1 -18425.347,E2 -18425.347} C_VEL
LIN {X 0,Y 262.644,Z 363.026,A -85,B 0,C 180,E1 -18427.585,E2 -18427.585} C_VEL
LIN {X 0,Y 260.323,Z 371.621,A -85,B 0,C 180,E1 -18429.866,E2 -18429.866} C_VEL
LIN {X 0,Y 258.213,Z 379.853,A -85,B 0,C 180,E1 -18432.578,E2 -18432.578} C_VEL
LIN {X 0,Y 256.729,Z 385.622,A -85,B 0,C 180,E1 -18434.926,E2 -18434.926} C_VEL
LIN {X 0,Y 255.472,Z 390.345,A -85,B 0,C 180,E1 -18437.286,E2 -18437.286} C_VEL
LIN {X 0,Y 254.551,Z 395.247,A -85,B 0,C 180,E1 -18440.464,E2 -18440.464} C_VEL
LIN {X 0,Y 254.055,Z 398.656,A -85,B 0,C 180,E1 -18443.647,E2 -18443.647} C_VEL
LIN {X 0,Y 253.911,Z 400.672,A -85,B 0,C 180,E1 -18446.826,E2 -18446.826} C_VEL
LIN {X 0,Y 254.011,Z 401.339,A -85,B 0,C 180,E1 -18450,E2 -18450} C_VEL
LIN {X 0,Y 253.906,Z 400.659,A -85,B 0,C 180,E1 -18453.173,E2 -18453.173} C_VEL
LIN {X 0,Y 254.054,Z 398.631,A -85,B 0,C 180,E1 -18456.353,E2 -18456.353} C_VEL
LIN {X 0,Y 254.545,Z 395.207,A -85,B 0,C 180,E1 -18459.535,E2 -18459.535} C_VEL
LIN {X 0,Y 255.47,Z 390.285,A -85,B 0,C 180,E1 -18462.714,E2 -18462.714} C_VEL
LIN {X 0,Y 256.725,Z 385.546,A -85,B 0,C 180,E1 -18465.074,E2 -18465.074} C_VEL
LIN {X 0,Y 258.37,Z 378.681,A -85,B 0,C 180,E1 -18467.816,E2 -18467.816} C_VEL
LIN {X 0,Y 260.658,Z 370.148,A -85,B 0,C 180,E1 -18470.519,E2 -18470.519} C_VEL
LIN {X 0,Y 263.083,Z 361.257,A -85,B 0,C 180,E1 -18472.79,E2 -18472.79} C_VEL
LIN {X 0,Y 265.359,Z 352.444,A -85,B 0,C 180,E1 -18474.654,E2 -18474.654} C_VEL
LIN {X 0,Y 267.997,Z 341.945,A -85,B 0,C 180,E1 -18476.475,E2 -18476.475} C_VEL
LIN {X 0,Y 270.462,Z 330.518,A -85,B 0,C 180,E1 -18478.098,E2 -18478.098} C_VEL
LIN {X 0,Y 269.537,Z 318.256,A -85,B 0,C 180,E1 -18479.872,E2 -18479.872} C_VEL
LIN {X 0,Y 267.48,Z 305.009,A -85,B 0,C 180,E1 -18481.586,E2 -18481.586} C_VEL
LIN {X 0,Y 264.612,Z 292.702,A -85,B 0,C 180,E1 -18483.037,E2 -18483.037} C_VEL
LIN {X 0,Y 260.576,Z 280.066,A -85,B 0,C 180,E1 -18484.441,E2 -18484.441} C_VEL
LIN {X 0,Y 257.076,Z 270.868,A -85,B 0,C 180,E1 -18485.402,E2 -18485.402} C_VEL
LIN {X 0,Y 256.936,Z 269.911,A -85,B 0,C 180,E1 -18485.493,E2 -18485.493} C_VEL
LIN {X 0,Y 257.397,Z 266.552,A -85,B 0,C 180,E1 -18488.902,E2 -18488.902} C_VEL
LIN {X 0,Y 257.457,Z 264.657,A -85,B 0,C 180,E1 -18490.931,E2 -18490.931} C_VEL
LIN {X 0,Y 257.375,Z 262.73,A -85,B 0,C 180,E1 -18493.052,E2 -18493.052} C_VEL
LIN {X 0,Y 256.919,Z 259.534,A -85,B 0,C 180,E1 -18496.853,E2 -18496.853} C_VEL
LIN {X 0,Y 256.464,Z 256.34,A -85,B 0,C 180,E1 -18500.929,E2 -18500.929} C_VEL
LIN {X 0,Y 256.252,Z 254.904,A -85,B 0,C 180,E1 -18502.888,E2 -18502.888} C_VEL
LIN {X 0,Y 256.105,Z 254.213,A -85,B 0,C 180,E1 -18505.412,E2 -18505.412} C_VEL
LIN {X 0,Y 256.083,Z 254.214,A -85,B 0,C 180,E1 -18508.571,E2 -18508.571} C_VEL
LIN {X 0,Y 256.094,Z 254.211,A -85,B 0,C 180,E1 -18512.191,E2 -18512.191} C_VEL
LIN {X 0,Y 256.134,Z 254.206,A -85,B 0,C 180,E1 -18515.696,E2 -18515.696} C_VEL
LIN {X 0,Y 256.15,Z 254.205,A -85,B 0,C 180,E1 -18519.104,E2 -18519.104} C_VEL
LIN {X 0,Y 256.249,Z 254.191,A -85,B 0,C 180,E1 -18524.082,E2 -18524.082} C_VEL
LIN {X 0,Y 256.289,Z 254.187,A -85,B 0,C 180,E1 -18527.328,E2 -18527.328} C_VEL
LIN {X 0,Y 256.435,Z 254.166,A -85,B 0,C 180,E1 -18530.623,E2 -18530.623} C_VEL
LIN {X 0,Y 256.46,Z 254.166,A -85,B 0,C 180,E1 -18533.707,E2 -18533.707} C_VEL
LIN {X 0,Y 256.714,Z 254.134,A -85,B 0,C 180,E1 -18538.431,E2 -18538.431} C_VEL
LIN {X 0,Y 256.712,Z 254.132,A -85,B 0,C 180,E1 -18541.569,E2 -18541.569} C_VEL
LIN {X 0,Y 256.471,Z 254.161,A -85,B 0,C 180,E1 -18546.762,E2 -18546.762} C_VEL
LIN {X 0,Y 256.428,Z 254.167,A -85,B 0,C 180,E1 -18549.465,E2 -18549.465} C_VEL
LIN {X 0,Y 256.257,Z 254.189,A -85,B 0,C 180,E1 -18554.29,E2 -18554.29} C_VEL
LIN {X 0,Y 256.212,Z 254.196,A -85,B 0,C 180,E1 -18557.562,E2 -18557.562} C_VEL
LIN {X 0,Y 256.155,Z 254.204,A -85,B 0,C 180,E1 -18561.118,E2 -18561.118} C_VEL
LIN {X 0,Y 256.172,Z 254.2,A -85,B 0,C 180,E1 -18565.13,E2 -18565.13} C_VEL
LIN {X 0,Y 256.105,Z 254.208,A -85,B 0,C 180,E1 -18569.601,E2 -18569.601} C_VEL
LIN {X 0,Y 256.069,Z 254.213,A -85,B 0,C 180,E1 -18573.293,E2 -18573.293} C_VEL
LIN {X 0,Y 256.111,Z 254.209,A -85,B 0,C 180,E1 -18577.269,E2 -18577.269} C_VEL
LIN {X 0,Y 256.063,Z 254.216,A -85,B 0,C 180,E1 -18582.179,E2 -18582.179} C_VEL
LIN {X 0,Y 256.085,Z 254.395,A -85,B 0,C 180,E1 -18583.322,E2 -18583.322} C_VEL
LIN {X 0,Y 256.488,Z 257.375,A -85,B 0,C 180,E1 -18587.717,E2 -18587.717} C_VEL
LIN {X 0,Y 256.572,Z 259.725,A -85,B 0,C 180,E1 -18590.949,E2 -18590.949} C_VEL
LIN {X 0,Y 256.363,Z 262.501,A -85,B 0,C 180,E1 -18594.489,E2 -18594.489} C_VEL
LIN {X 0,Y 257.483,Z 265.797,A -85,B 0,C 180,E1 -18594.823,E2 -18594.823} C_VEL
LIN {X 0,Y 262.165,Z 277.07,A -85,B 0,C 180,E1 -18596.149,E2 -18596.149} C_VEL
LIN {X 0,Y 266.207,Z 289.471,A -85,B 0,C 180,E1 -18597.653,E2 -18597.653} C_VEL
LIN {X 0,Y 269.062,Z 300.705,A -85,B 0,C 180,E1 -18599.109,E2 -18599.109} C_VEL
LIN {X 0,Y 271.112,Z 311.938,A -85,B 0,C 180,E1 -18600.683,E2 -18600.683} C_VEL
LIN {X 0,Y 271.799,Z 317.674,A -85,B 0,C 180,E1 -18601.54,E2 -18601.54} C_VEL
LIN {X 0,Y 270.526,Z 325.208,A -85,B 0,C 180,E1 -18602.54,E2 -18602.54} C_VEL
LIN {X 0,Y 267.814,Z 336.995,A -85,B 0,C 180,E1 -18604.342,E2 -18604.342} C_VEL
LIN {X 0,Y 265.351,Z 346.752,A -85,B 0,C 180,E1 -18606.177,E2 -18606.177} C_VEL
LIN {X 0,Y 262.709,Z 356.493,A -85,B 0,C 180,E1 -18608.418,E2 -18608.418} C_VEL
LIN {X 0,Y 260.152,Z 365.55,A -85,B 0,C 180,E1 -18611.002,E2 -18611.002} C_VEL
LIN {X 0,Y 258.501,Z 372.297,A -85,B 0,C 180,E1 -18613.413,E2 -18613.413} C_VEL
LIN {X 0,Y 256.858,Z 377.697,A -85,B 0,C 180,E1 -18615.744,E2 -18615.744} C_VEL
LIN {X 0,Y 255.506,Z 383.366,A -85,B 0,C 180,E1 -18618.899,E2 -18618.899} C_VEL
LIN {X 0,Y 254.615,Z 387.484,A -85,B 0,C 180,E1 -18622.067,E2 -18622.067} C_VEL
LIN {X 0,Y 254.159,Z 390.174,A -85,B 0,C 180,E1 -18625.242,E2 -18625.242} C_VEL
LIN {X 0,Y 254.001,Z 391.519,A -85,B 0,C 180,E1 -18628.415,E2 -18628.415} C_VEL
LIN {X 0,Y 254.001,Z 391.547,A -85,B 0,C 180,E1 -18631.586,E2 -18631.586} C_VEL
LIN {X 0,Y 254.153,Z 390.257,A -85,B 0,C 180,E1 -18634.759,E2 -18634.759} C_VEL
LIN {X 0,Y 254.614,Z 387.616,A -85,B 0,C 180,E1 -18637.933,E2 -18637.933} C_VEL
LIN {X 0,Y 255.475,Z 383.556,A -85,B 0,C 180,E1 -18641.103,E2 -18641.103} C_VEL
LIN {X 0,Y 256.813,Z 377.945,A -85,B 0,C 180,E1 -18644.259,E2 -18644.259} C_VEL
LIN {X 0,Y 258.757,Z 371.6,A -85,B 0,C 180,E1 -18646.977,E2 -18646.977} C_VEL
LIN {X 0,Y 260.347,Z 364.945,A -85,B 0,C 180,E1 -18649.311,E2 -18649.311} C_VEL
LIN {X 0,Y 262.638,Z 356.944,A -85,B 0,C 180,E1 -18651.589,E2 -18651.589} C_VEL
LIN {X 0,Y 265.254,Z 347.291,A -85,B 0,C 180,E1 -18653.832,E2 -18653.832} C_VEL
LIN {X 0,Y 267.998,Z 336.575,A -85,B 0,C 180,E1 -18655.848,E2 -18655.848} C_VEL
LIN {X 0,Y 270.703,Z 324.695,A -85,B 0,C 180,E1 -18657.65,E2 -18657.65} C_VEL
LIN {X 0,Y 271.891,Z 318.222,A -85,B 0,C 180,E1 -18658.495,E2 -18658.495} C_VEL
LIN {X 0,Y 270.385,Z 307.118,A -85,B 0,C 180,E1 -18660.128,E2 -18660.128} C_VEL
LIN {X 0,Y 267.771,Z 294.844,A -85,B 0,C 180,E1 -18661.783,E2 -18661.783} C_VEL
LIN {X 0,Y 263.956,Z 282.122,A -85,B 0,C 180,E1 -18663.382,E2 -18663.382} C_VEL
LIN {X 0,Y 259.49,Z 270.197,A -85,B 0,C 180,E1 -18664.788,E2 -18664.788} C_VEL
LIN {X 0,Y 256.591,Z 263.668,A -85,B 0,C 180,E1 -18665.543,E2 -18665.543} C_VEL
LIN {X 0,Y 256.366,Z 262.48,A -85,B 0,C 180,E1 -18665.68,E2 -18665.68} C_VEL
LIN {X 0,Y 256.568,Z 259.827,A -85,B 0,C 180,E1 -18669.052,E2 -18669.052} C_VEL
LIN {X 0,Y 256.489,Z 257.45,A -85,B 0,C 180,E1 -18672.284,E2 -18672.284} C_VEL
LIN {X 0,Y 256.086,Z 254.503,A -85,B 0,C 180,E1 -18676.678,E2 -18676.678} C_VEL
LIN {X 0,Y 256.042,Z 254.219,A -85,B 0,C 180,E1 -18678.794,E2 -18678.794} C_VEL
LIN {X 0,Y 256.128,Z 254.207,A -85,B 0,C 180,E1 -18682.867,E2 -18682.867} C_VEL
LIN {X 0,Y 256.07,Z 254.213,A -85,B 0,C 180,E1 -18686.707,E2 -18686.707} C_VEL
LIN {X 0,Y 256.116,Z 254.208,A -85,B 0,C 180,E1 -18690.4,E2 -18690.4} C_VEL
LIN {X 0,Y 256.173,Z 254.194,A -85,B 0,C 180,E1 -18694.87,E2 -18694.87} C_VEL
LIN {X 0,Y 256.166,Z 254.202,A -85,B 0,C 180,E1 -18699.105,E2 -18699.105} C_VEL
LIN {X 0,Y 256.303,Z 254.183,A -85,B 0,C 180,E1 -18704.085,E2 -18704.085} C_VEL
LIN {X 0,Y 256.298,Z 254.183,A -85,B 0,C 180,E1 -18708.933,E2 -18708.933} C_VEL
LIN {X 0,Y 256.507,Z 254.157,A -85,B 0,C 180,E1 -18712.126,E2 -18712.126} C_VEL
LIN {X 0,Y 256.496,Z 254.159,A -85,B 0,C 180,E1 -18716.858,E2 -18716.858} C_VEL
LIN {X 0,Y 256.71,Z 254.135,A -85,B 0,C 180,E1 -18718.431,E2 -18718.431} C_VEL
LIN {X 0,Y 256.716,Z 254.134,A -85,B 0,C 180,E1 -18721.569,E2 -18721.569} C_VEL
LIN {X 0,Y 256.461,Z 254.165,A -85,B 0,C 180,E1 -18726.293,E2 -18726.293} C_VEL
LIN {X 0,Y 256.429,Z 254.169,A -85,B 0,C 180,E1 -18729.465,E2 -18729.465} C_VEL
LIN {X 0,Y 256.238,Z 254.193,A -85,B 0,C 180,E1 -18734.291,E2 -18734.291} C_VEL
LIN {X 0,Y 256.183,Z 254.2,A -85,B 0,C 180,E1 -18737.564,E2 -18737.564} C_VEL
LIN {X 0,Y 256.144,Z 254.204,A -85,B 0,C 180,E1 -18741.111,E2 -18741.111} C_VEL
LIN {X 0,Y 256.079,Z 254.211,A -85,B 0,C 180,E1 -18742.356,E2 -18742.356} C_VEL
LIN {X 0,Y 255.423,Z 254.298,A -85,B 0,C 180,E1 -18743.669,E2 -18743.669} C_VEL
LIN {X 0,Y 252.601,Z 254.654,A -85,B 0,C 180,E1 -18745.811,E2 -18745.811} C_VEL
LIN {X 0,Y 250.182,Z 254.952,A -85,B 0,C 180,E1 -18747.554,E2 -18747.554} C_VEL
LIN {X 0,Y 249.115,Z 255.08,A -85,B 0,C 180,E1 -18748.905,E2 -18748.905} C_VEL
LIN {X 0,Y 249.013,Z 255.091,A -85,B 0,C 180,E1 -18749.363,E2 -18749.363} C_VEL
LIN {X 0,Y 249.029,Z 255.092,A -85,B 0,C 180,E1 -18752.426,E2 -18752.426} C_VEL
LIN {X 0,Y 249.047,Z 255.092,A -85,B 0,C 180,E1 -18755.078,E2 -18755.078} C_VEL
LIN {X 0,Y 249.432,Z 257.156,A -85,B 0,C 180,E1 -18758.307,E2 -18758.307} C_VEL
LIN {X 0,Y 249.889,Z 260.272,A -85,B 0,C 180,E1 -18762.453,E2 -18762.453} C_VEL
LIN {X 0,Y 250.258,Z 262.631,A -85,B 0,C 180,E1 -18765.406,E2 -18765.406} C_VEL
LIN {X 0,Y 250.477,Z 265.942,A -85,B 0,C 180,E1 -18769.251,E2 -18769.251} C_VEL
LIN {X 0,Y 250.33,Z 268.356,A -85,B 0,C 180,E1 -18771.855,E2 -18771.855} C_VEL
LIN {X 0,Y 250.115,Z 269.955,A -85,B 0,C 180,E1 -18773.374,E2 -18773.374} C_VEL
LIN {X 0,Y 251.237,Z 273.333,A -85,B 0,C 180,E1 -18773.703,E2 -18773.703} C_VEL
LIN {X 0,Y 255.817,Z 285.555,A -85,B 0,C 180,E1 -18775.12,E2 -18775.12} C_VEL
LIN {X 0,Y 259.231,Z 297.444,A -85,B 0,C 180,E1 -18776.543,E2 -18776.543} C_VEL
LIN {X 0,Y 261.474,Z 307.774,A -85,B 0,C 180,E1 -18777.85,E2 -18777.85} C_VEL
LIN {X 0,Y 263.285,Z 320.87,A -85,B 0,C 180,E1 -18779.654,E2 -18779.654} C_VEL
LIN {X 0,Y 263.91,Z 330.626,A -85,B 0,C 180,E1 -18781.139,E2 -18781.139} C_VEL
LIN {X 0,Y 263.539,Z 333.629,A -85,B 0,C 180,E1 -18781.574,E2 -18781.574} C_VEL
LIN {X 0,Y 260.838,Z 345.35,A -85,B 0,C 180,E1 -18783.388,E2 -18783.388} C_VEL
LIN {X 0,Y 257.907,Z 356.157,A -85,B 0,C 180,E1 -18785.445,E2 -18785.445} C_VEL
LIN {X 0,Y 255.196,Z 365.901,A -85,B 0,C 180,E1 -18787.748,E2 -18787.748} C_VEL
LIN {X 0,Y 252.918,Z 373.988,A -85,B 0,C 180,E1 -18790.099,E2 -18790.099} C_VEL
LIN {X 0,Y 250.886,Z 381.745,A -85,B 0,C 180,E1 -18792.894,E2 -18792.894} C_VEL
LIN {X 0,Y 249.368,Z 387.157,A -85,B 0,C 180,E1 -18795.306,E2 -18795.306} C_VEL
LIN {X 0,Y 247.945,Z 392.856,A -85,B 0,C 180,E1 -18798.556,E2 -18798.556} C_VEL
LIN {X 0,Y 247.183,Z 396.995,A -85,B 0,C 180,E1 -18801.827,E2 -18801.827} C_VEL
LIN {X 0,Y 246.882,Z 399.7,A -85,B 0,C 180,E1 -18805.101,E2 -18805.101} C_VEL
LIN {X 0,Y 246.858,Z 401.039,A -85,B 0,C 180,E1 -18808.368,E2 -18808.368} C_VEL
LIN {X 0,Y 246.919,Z 401.204,A -85,B 0,C 180,E1 -18810,E2 -18810} C_VEL
LIN {X 0,Y 246.811,Z 400.523,A -85,B 0,C 180,E1 -18813.265,E2 -18813.265} C_VEL
LIN {X 0,Y 246.974,Z 398.495,A -85,B 0,C 180,E1 -18816.536,E2 -18816.536} C_VEL
LIN {X 0,Y 247.519,Z 395.071,A -85,B 0,C 180,E1 -18819.809,E2 -18819.809} C_VEL
LIN {X 0,Y 248.507,Z 390.148,A -85,B 0,C 180,E1 -18823.076,E2 -18823.076} C_VEL
LIN {X 0,Y 249.836,Z 385.409,A -85,B 0,C 180,E1 -18825.5,E2 -18825.5} C_VEL
LIN {X 0,Y 251.446,Z 379.039,A -85,B 0,C 180,E1 -18828.138,E2 -18828.138} C_VEL
LIN {X 0,Y 253.609,Z 371.369,A -85,B 0,C 180,E1 -18830.691,E2 -18830.691} C_VEL
LIN {X 0,Y 256.059,Z 362.75,A -85,B 0,C 180,E1 -18833.024,E2 -18833.024} C_VEL
LIN {X 0,Y 258.907,Z 352.306,A -85,B 0,C 180,E1 -18835.311,E2 -18835.311} C_VEL
LIN {X 0,Y 261.636,Z 341.806,A -85,B 0,C 180,E1 -18837.171,E2 -18837.171} C_VEL
LIN {X 0,Y 263.92,Z 331.807,A -85,B 0,C 180,E1 -18838.641,E2 -18838.641} C_VEL
LIN {X 0,Y 263.14,Z 319.559,A -85,B 0,C 180,E1 -18840.495,E2 -18840.495} C_VEL
LIN {X 0,Y 261.035,Z 305.679,A -85,B 0,C 180,E1 -18842.377,E2 -18842.377} C_VEL
LIN {X 0,Y 258.607,Z 295.106,A -85,B 0,C 180,E1 -18843.709,E2 -18843.709} C_VEL
LIN {X 0,Y 255.017,Z 283.35,A -85,B 0,C 180,E1 -18845.1,E2 -18845.1} C_VEL
LIN {X 0,Y 251.036,Z 272.963,A -85,B 0,C 180,E1 -18846.295,E2 -18846.295} C_VEL
LIN {X 0,Y 250.082,Z 269.746,A -85,B 0,C 180,E1 -18846.645,E2 -18846.645} C_VEL
LIN {X 0,Y 250.47,Z 266.4,A -85,B 0,C 180,E1 -18850.193,E2 -18850.193} C_VEL
LIN {X 0,Y 250.376,Z 263.807,A -85,B 0,C 180,E1 -18853.129,E2 -18853.129} C_VEL
LIN {X 0,Y 249.879,Z 260.224,A -85,B 0,C 180,E1 -18857.545,E2 -18857.545} C_VEL
LIN {X 0,Y 249.384,Z 256.808,A -85,B 0,C 180,E1 -18862.1,E2 -18862.1} C_VEL
LIN {X 0,Y 249.046,Z 255.092,A -85,B 0,C 180,E1 -18864.922,E2 -18864.922} C_VEL
LIN {X 0,Y 249.002,Z 255.095,A -85,B 0,C 180,E1 -18869.466,E2 -18869.466} C_VEL
LIN {X 0,Y 249.036,Z 255.089,A -85,B 0,C 180,E1 -18873.158,E2 -18873.158} C_VEL
LIN {X 0,Y 249.056,Z 255.088,A -85,B 0,C 180,E1 -18876.73,E2 -18876.73} C_VEL
LIN {X 0,Y 249.089,Z 255.083,A -85,B 0,C 180,E1 -18880.21,E2 -18880.21} C_VEL
LIN {X 0,Y 249.196,Z 255.069,A -85,B 0,C 180,E1 -18883.619,E2 -18883.619} C_VEL
LIN {X 0,Y 249.243,Z 255.059,A -85,B 0,C 180,E1 -18888.616,E2 -18888.616} C_VEL
LIN {X 0,Y 249.436,Z 255.04,A -85,B 0,C 180,E1 -18891.901,E2 -18891.901} C_VEL
LIN {X 0,Y 249.431,Z 255.039,A -85,B 0,C 180,E1 -18896.77,E2 -18896.77} C_VEL
LIN {X 0,Y 249.676,Z 255.011,A -85,B 0,C 180,E1 -18898.387,E2 -18898.387} C_VEL
LIN {X 0,Y 249.674,Z 255.009,A -85,B 0,C 180,E1 -18901.613,E2 -18901.613} C_VEL
LIN {X 0,Y 249.44,Z 255.037,A -85,B 0,C 180,E1 -18906.748,E2 -18906.748} C_VEL
LIN {X 0,Y 249.345,Z 255.051,A -85,B 0,C 180,E1 -18909.737,E2 -18909.737} C_VEL
LIN {X 0,Y 249.207,Z 255.07,A -85,B 0,C 180,E1 -18914.703,E2 -18914.703} C_VEL
LIN {X 0,Y 249.141,Z 255.076,A -85,B 0,C 180,E1 -18918.077,E2 -18918.077} C_VEL
LIN {X 0,Y 249.086,Z 255.082,A -85,B 0,C 180,E1 -18921.518,E2 -18921.518} C_VEL
LIN {X 0,Y 249.119,Z 255.079,A -85,B 0,C 180,E1 -18925.476,E2 -18925.476} C_VEL
LIN {X 0,Y 249.075,Z 255.084,A -85,B 0,C 180,E1 -18928.989,E2 -18928.989} C_VEL
LIN {X 0,Y 249.032,Z 255.09,A -85,B 0,C 180,E1 -18932.426,E2 -18932.426} C_VEL
LIN {X 0,Y 249.027,Z 255.091,A -85,B 0,C 180,E1 -18936.346,E2 -18936.346} C_VEL
LIN {X 0,Y 248.985,Z 255.097,A -85,B 0,C 180,E1 -18940.482,E2 -18940.482} C_VEL
LIN {X 0,Y 249.035,Z 255.321,A -85,B 0,C 180,E1 -18942.799,E2 -18942.799} C_VEL
LIN {X 0,Y 249.276,Z 256.833,A -85,B 0,C 180,E1 -18945.183,E2 -18945.183} C_VEL
LIN {X 0,Y 249.476,Z 258.357,A -85,B 0,C 180,E1 -18947.46,E2 -18947.46} C_VEL
LIN {X 0,Y 249.572,Z 259.898,A -85,B 0,C 180,E1 -18949.633,E2 -18949.633} C_VEL
LIN {X 0,Y 249.431,Z 262.775,A -85,B 0,C 180,E1 -18953.373,E2 -18953.373} C_VEL
LIN {X 0,Y 250.495,Z 265.852,A -85,B 0,C 180,E1 -18953.683,E2 -18953.683} C_VEL
LIN {X 0,Y 251.686,Z 268.322,A -85,B 0,C 180,E1 -18953.999,E2 -18953.999} C_VEL
LIN {X 0,Y 256.394,Z 279.816,A -85,B 0,C 180,E1 -18955.45,E2 -18955.45} C_VEL
LIN {X 0,Y 260.521,Z 293.065,A -85,B 0,C 180,E1 -18957.165,E2 -18957.165} C_VEL
LIN {X 0,Y 263.137,Z 304.28,A -85,B 0,C 180,E1 -18958.724,E2 -18958.724} C_VEL
LIN {X 0,Y 265.108,Z 316.854,A -85,B 0,C 180,E1 -18960.616,E2 -18960.616} C_VEL
LIN {X 0,Y 265.184,Z 320.848,A -85,B 0,C 180,E1 -18961.226,E2 -18961.226} C_VEL
LIN {X 0,Y 262.51,Z 332.709,A -85,B 0,C 180,E1 -18962.927,E2 -18962.927} C_VEL
LIN {X 0,Y 259.851,Z 343.199,A -85,B 0,C 180,E1 -18964.787,E2 -18964.787} C_VEL
LIN {X 0,Y 257.018,Z 353.615,A -85,B 0,C 180,E1 -18967.067,E2 -18967.067} C_VEL
LIN {X 0,Y 254.456,Z 362.204,A -85,B 0,C 180,E1 -18969.381,E2 -18969.381} C_VEL
LIN {X 0,Y 252.536,Z 368.928,A -85,B 0,C 180,E1 -18971.601,E2 -18971.601} C_VEL
LIN {X 0,Y 251.086,Z 374.361,A -85,B 0,C 180,E1 -18973.746,E2 -18973.746} C_VEL
LIN {X 0,Y 249.534,Z 379.436,A -85,B 0,C 180,E1 -18976.149,E2 -18976.149} C_VEL
LIN {X 0,Y 248.238,Z 384.689,A -85,B 0,C 180,E1 -18979.396,E2 -18979.396} C_VEL
LIN {X 0,Y 247.582,Z 387.62,A -85,B 0,C 180,E1 -18981.84,E2 -18981.84} C_VEL
LIN {X 0,Y 247.075,Z 390.31,A -85,B 0,C 180,E1 -18985.105,E2 -18985.105} C_VEL
LIN {X 0,Y 246.915,Z 391.653,A -85,B 0,C 180,E1 -18988.369,E2 -18988.369} C_VEL
LIN {X 0,Y 246.915,Z 391.682,A -85,B 0,C 180,E1 -18991.631,E2 -18991.631} C_VEL
LIN {X 0,Y 247.065,Z 390.392,A -85,B 0,C 180,E1 -18994.896,E2 -18994.896} C_VEL
LIN {X 0,Y 247.582,Z 387.75,A -85,B 0,C 180,E1 -18998.16,E2 -18998.16} C_VEL
LIN {X 0,Y 248.492,Z 383.69,A -85,B 0,C 180,E1 -19001.419,E2 -19001.419} C_VEL
LIN {X 0,Y 249.921,Z 378.079,A -85,B 0,C 180,E1 -19004.661,E2 -19004.661} C_VEL
LIN {X 0,Y 251.942,Z 371.734,A -85,B 0,C 180,E1 -19007.45,E2 -19007.45} C_VEL
LIN {X 0,Y 253.648,Z 365.078,A -85,B 0,C 180,E1 -19009.842,E2 -19009.842} C_VEL
LIN {X 0,Y 256.03,Z 357.077,A -85,B 0,C 180,E1 -19012.175,E2 -19012.175} C_VEL
LIN {X 0,Y 258.746,Z 347.424,A -85,B 0,C 180,E1 -19014.47,E2 -19014.47} C_VEL
LIN {X 0,Y 261.622,Z 336.706,A -85,B 0,C 180,E1 -19016.526,E2 -19016.526} C_VEL
LIN {X 0,Y 264.429,Z 324.826,A -85,B 0,C 180,E1 -19018.365,E2 -19018.365} C_VEL
LIN {X 0,Y 265.388,Z 319.505,A -85,B 0,C 180,E1 -19019.084,E2 -19019.084} C_VEL
LIN {X 0,Y 263.875,Z 307.929,A -85,B 0,C 180,E1 -19020.867,E2 -19020.867} C_VEL
LIN {X 0,Y 261.403,Z 296.194,A -85,B 0,C 180,E1 -19022.528,E2 -19022.528} C_VEL
LIN {X 0,Y 257.498,Z 282.959,A -85,B 0,C 180,E1 -19024.28,E2 -19024.28} C_VEL
LIN {X 0,Y 252.735,Z 270.518,A -85,B 0,C 180,E1 -19025.849,E2 -19025.849} C_VEL
LIN {X 0,Y 250.486,Z 265.813,A -85,B 0,C 180,E1 -19026.463,E2 -19026.463} C_VEL
LIN {X 0,Y 249.44,Z 262.623,A -85,B 0,C 180,E1 -19026.812,E2 -19026.812} C_VEL
LIN {X 0,Y 249.555,Z 259.879,A -85,B 0,C 180,E1 -19030.502,E2 -19030.502} C_VEL
LIN {X 0,Y 249.43,Z 258.226,A -85,B 0,C 180,E1 -19032.896,E2 -19032.896} C_VEL
LIN {X 0,Y 249.035,Z 255.426,A -85,B 0,C 180,E1 -19037.202,E2 -19037.202} C_VEL
LIN {X 0,Y 248.988,Z 255.095,A -85,B 0,C 180,E1 -19039.651,E2 -19039.651} C_VEL
LIN {X 0,Y 249.028,Z 255.091,A -85,B 0,C 180,E1 -19043.654,E2 -19043.654} C_VEL
LIN {X 0,Y 249.04,Z 255.089,A -85,B 0,C 180,E1 -19047.846,E2 -19047.846} C_VEL
LIN {X 0,Y 249.099,Z 255.082,A -85,B 0,C 180,E1 -19051.338,E2 -19051.338} C_VEL
LIN {X 0,Y 249.137,Z 255.07,A -85,B 0,C 180,E1 -19054.967,E2 -19054.967} C_VEL
LIN {X 0,Y 249.112,Z 255.078,A -85,B 0,C 180,E1 -19060.211,E2 -19060.211} C_VEL
LIN {X 0,Y 249.245,Z 255.064,A -85,B 0,C 180,E1 -19063.622,E2 -19063.622} C_VEL
LIN {X 0,Y 249.246,Z 255.063,A -85,B 0,C 180,E1 -19068.616,E2 -19068.616} C_VEL
LIN {X 0,Y 249.449,Z 255.036,A -85,B 0,C 180,E1 -19071.902,E2 -19071.902} C_VEL
LIN {X 0,Y 249.291,Z 255.056,A -85,B 0,C 180,E1 -19075.148,E2 -19075.148} C_VEL
LIN {X 0,Y 249.672,Z 255.011,A -85,B 0,C 180,E1 -19078.387,E2 -19078.387} C_VEL
LIN {X 0,Y 249.677,Z 255.01,A -85,B 0,C 180,E1 -19081.613,E2 -19081.613} C_VEL
LIN {X 0,Y 249.434,Z 255.041,A -85,B 0,C 180,E1 -19086.471,E2 -19086.471} C_VEL
LIN {X 0,Y 249.345,Z 255.05,A -85,B 0,C 180,E1 -19089.736,E2 -19089.736} C_VEL
LIN {X 0,Y 249.181,Z 255.071,A -85,B 0,C 180,E1 -19094.705,E2 -19094.705} C_VEL
LIN {X 0,Y 249.118,Z 255.08,A -85,B 0,C 180,E1 -19098.079,E2 -19098.079} C_VEL
LIN {X 0,Y 249.041,Z 255.085,A -85,B 0,C 180,E1 -19102.349,E2 -19102.349} C_VEL
LIN {X 0,Y 249.087,Z 255.076,A -85,B 0,C 180,E1 -19105.46,E2 -19105.46} C_VEL
LIN {X 0,Y 249.013,Z 255.091,A -85,B 0,C 180,E1 -19109.363,E2 -19109.363} C_VEL
LIN {X 0,Y 248.299,Z 255.181,A -85,B 0,C 180,E1 -19110.713,E2 -19110.713} C_VEL
LIN {X 0,Y 245.449,Z 255.586,A -85,B 0,C 180,E1 -19112.916,E2 -19112.916} C_VEL
LIN {X 0,Y 243.125,Z 256.265,A -85,B 0,C 180,E1 -19114.704,E2 -19114.704} C_VEL
LIN {X 0,Y 242.222,Z 257.007,A -85,B 0,C 180,E1 -19116.083,E2 -19116.083} C_VEL
LIN {X 0,Y 242.197,Z 257.303,A -85,B 0,C 180,E1 -19116.548,E2 -19116.548} C_VEL
LIN {X 0,Y 242.561,Z 259.408,A -85,B 0,C 180,E1 -19119.601,E2 -19119.601} C_VEL
LIN {X 0,Y 243.071,Z 262.661,A -85,B 0,C 180,E1 -19123.941,E2 -19123.941} C_VEL
LIN {X 0,Y 243.324,Z 264.483,A -85,B 0,C 180,E1 -19126.227,E2 -19126.227} C_VEL
LIN {X 0,Y 243.42,Z 266.507,A -85,B 0,C 180,E1 -19128.648,E2 -19128.648} C_VEL
LIN {X 0,Y 243.247,Z 269.647,A -85,B 0,C 180,E1 -19132.155,E2 -19132.155} C_VEL
LIN {X 0,Y 244.175,Z 272.774,A -85,B 0,C 180,E1 -19132.458,E2 -19132.458} C_VEL
LIN {X 0,Y 245.376,Z 275.47,A -85,B 0,C 180,E1 -19132.796,E2 -19132.796} C_VEL
LIN {X 0,Y 249.731,Z 287.262,A -85,B 0,C 180,E1 -19134.265,E2 -19134.265} C_VEL
LIN {X 0,Y 252.754,Z 297.871,A -85,B 0,C 180,E1 -19135.619,E2 -19135.619} C_VEL
LIN {X 0,Y 255.341,Z 310.189,A -85,B 0,C 180,E1 -19137.276,E2 -19137.276} C_VEL
LIN {X 0,Y 256.978,Z 323.684,A -85,B 0,C 180,E1 -19139.25,E2 -19139.25} C_VEL
LIN {X 0,Y 257.426,Z 331.919,A -85,B 0,C 180,E1 -19140.566,E2 -19140.566} C_VEL
LIN {X 0,Y 255.345,Z 341.885,A -85,B 0,C 180,E1 -19142.102,E2 -19142.102} C_VEL
LIN {X 0,Y 252.501,Z 352.347,A -85,B 0,C 180,E1 -19143.999,E2 -19143.999} C_VEL
LIN {X 0,Y 249.959,Z 361.128,A -85,B 0,C 180,E1 -19145.94,E2 -19145.94} C_VEL
LIN {X 0,Y 247.338,Z 369.995,A -85,B 0,C 180,E1 -19148.322,E2 -19148.322} C_VEL
LIN {X 0,Y 245.188,Z 377.38,A -85,B 0,C 180,E1 -19150.754,E2 -19150.754} C_VEL
LIN {X 0,Y 243.458,Z 383.535,A -85,B 0,C 180,E1 -19153.221,E2 -19153.221} C_VEL
LIN {X 0,Y 242.018,Z 388.638,A -85,B 0,C 180,E1 -19155.71,E2 -19155.71} C_VEL
LIN {X 0,Y 240.695,Z 393.906,A -85,B 0,C 180,E1 -19159.059,E2 -19159.059} C_VEL
LIN {X 0,Y 240.141,Z 396.861,A -85,B 0,C 180,E1 -19161.585,E2 -19161.585} C_VEL
LIN {X 0,Y 239.799,Z 399.566,A -85,B 0,C 180,E1 -19164.956,E2 -19164.956} C_VEL
LIN {X 0,Y 239.771,Z 400.904,A -85,B 0,C 180,E1 -19168.32,E2 -19168.32} C_VEL
LIN {X 0,Y 239.83,Z 401.069,A -85,B 0,C 180,E1 -19170,E2 -19170} C_VEL
LIN {X 0,Y 239.72,Z 400.388,A -85,B 0,C 180,E1 -19173.361,E2 -19173.361} C_VEL
LIN {X 0,Y 239.896,Z 398.359,A -85,B 0,C 180,E1 -19176.729,E2 -19176.729} C_VEL
LIN {X 0,Y 240.479,Z 394.934,A -85,B 0,C 180,E1 -19180.099,E2 -19180.099} C_VEL
LIN {X 0,Y 241.562,Z 390.012,A -85,B 0,C 180,E1 -19183.459,E2 -19183.459} C_VEL
LIN {X 0,Y 242.95,Z 385.272,A -85,B 0,C 180,E1 -19185.951,E2 -19185.951} C_VEL
LIN {X 0,Y 244.787,Z 378.512,A -85,B 0,C 180,E1 -19188.8,E2 -19188.8} C_VEL
LIN {X 0,Y 247.332,Z 369.873,A -85,B 0,C 180,E1 -19191.678,E2 -19191.678} C_VEL
LIN {X 0,Y 249.951,Z 360.98,A -85,B 0,C 180,E1 -19194.061,E2 -19194.061} C_VEL
LIN {X 0,Y 253.026,Z 350.212,A -85,B 0,C 180,E1 -19196.386,E2 -19196.386} C_VEL
LIN {X 0,Y 255.777,Z 339.704,A -85,B 0,C 180,E1 -19198.219,E2 -19198.219} C_VEL
LIN {X 0,Y 257.303,Z 333.389,A -85,B 0,C 180,E1 -19199.158,E2 -19199.158} C_VEL
LIN {X 0,Y 256.946,Z 323.523,A -85,B 0,C 180,E1 -19200.734,E2 -19200.734} C_VEL
LIN {X 0,Y 255.392,Z 311.092,A -85,B 0,C 180,E1 -19202.564,E2 -19202.564} C_VEL
LIN {X 0,Y 253.152,Z 299.652,A -85,B 0,C 180,E1 -19204.107,E2 -19204.107} C_VEL
LIN {X 0,Y 249.644,Z 287.113,A -85,B 0,C 180,E1 -19205.708,E2 -19205.708} C_VEL
LIN {X 0,Y 244.735,Z 273.795,A -85,B 0,C 180,E1 -19207.343,E2 -19207.343} C_VEL
LIN {X 0,Y 243.444,Z 271.015,A -85,B 0,C 180,E1 -19207.694,E2 -19207.694} C_VEL
LIN {X 0,Y 243.19,Z 269.63,A -85,B 0,C 180,E1 -19207.82,E2 -19207.82} C_VEL
LIN {X 0,Y 243.392,Z 266.237,A -85,B 0,C 180,E1 -19211.616,E2 -19211.616} C_VEL
LIN {X 0,Y 243.285,Z 264.34,A -85,B 0,C 180,E1 -19213.893,E2 -19213.893} C_VEL
LIN {X 0,Y 242.775,Z 260.918,A -85,B 0,C 180,E1 -19218.255,E2 -19218.255} C_VEL
LIN {X 0,Y 242.345,Z 257.884,A -85,B 0,C 180,E1 -19222.483,E2 -19222.483} C_VEL
LIN {X 0,Y 242.077,Z 256.549,A -85,B 0,C 180,E1 -19224.504,E2 -19224.504} C_VEL
LIN {X 0,Y 241.988,Z 255.971,A -85,B 0,C 180,E1 -19227.377,E2 -19227.377} C_VEL
LIN {X 0,Y 241.977,Z 255.97,A -85,B 0,C 180,E1 -19230.613,E2 -19230.613} C_VEL
LIN {X 0,Y 242.033,Z 255.963,A -85,B 0,C 180,E1 -19234.179,E2 -19234.179} C_VEL
LIN {X 0,Y 242.023,Z 255.964,A -85,B 0,C 180,E1 -19238.316,E2 -19238.316} C_VEL
LIN {X 0,Y 242.116,Z 255.95,A -85,B 0,C 180,E1 -19243.316,E2 -19243.316} C_VEL
LIN {X 0,Y 242.154,Z 255.944,A -85,B 0,C 180,E1 -19246.574,E2 -19246.574} C_VEL
LIN {X 0,Y 242.386,Z 255.919,A -85,B 0,C 180,E1 -19251.664,E2 -19251.664} C_VEL
LIN {X 0,Y 242.245,Z 255.934,A -85,B 0,C 180,E1 -19255.007,E2 -19255.007} C_VEL
LIN {X 0,Y 242.636,Z 255.888,A -85,B 0,C 180,E1 -19258.34,E2 -19258.34} C_VEL
LIN {X 0,Y 242.634,Z 255.886,A -85,B 0,C 180,E1 -19261.66,E2 -19261.66} C_VEL
LIN {X 0,Y 242.42,Z 255.912,A -85,B 0,C 180,E1 -19266.721,E2 -19266.721} C_VEL
LIN {X 0,Y 242.269,Z 255.933,A -85,B 0,C 180,E1 -19270.024,E2 -19270.024} C_VEL
LIN {X 0,Y 242.169,Z 255.945,A -85,B 0,C 180,E1 -19275.141,E2 -19275.141} C_VEL
LIN {X 0,Y 242.074,Z 255.956,A -85,B 0,C 180,E1 -19278.624,E2 -19278.624} C_VEL
LIN {X 0,Y 242.008,Z 255.963,A -85,B 0,C 180,E1 -19282.181,E2 -19282.181} C_VEL
LIN {X 0,Y 242.068,Z 255.956,A -85,B 0,C 180,E1 -19285.838,E2 -19285.838} C_VEL
LIN {X 0,Y 242.008,Z 255.964,A -85,B 0,C 180,E1 -19289.583,E2 -19289.583} C_VEL
LIN {X 0,Y 241.981,Z 255.969,A -85,B 0,C 180,E1 -19293.493,E2 -19293.493} C_VEL
LIN {X 0,Y 241.984,Z 255.969,A -85,B 0,C 180,E1 -19297.583,E2 -19297.583} C_VEL
LIN {X 0,Y 241.936,Z 256.071,A -85,B 0,C 180,E1 -19301.923,E2 -19301.923} C_VEL
LIN {X 0,Y 242.362,Z 258.879,A -85,B 0,C 180,E1 -19306.465,E2 -19306.465} C_VEL
LIN {X 0,Y 242.511,Z 261.569,A -85,B 0,C 180,E1 -19310.39,E2 -19310.39} C_VEL
LIN {X 0,Y 242.507,Z 262.954,A -85,B 0,C 180,E1 -19312.146,E2 -19312.146} C_VEL
LIN {X 0,Y 243.581,Z 265.977,A -85,B 0,C 180,E1 -19312.475,E2 -19312.475} C_VEL
LIN {X 0,Y 244.912,Z 268.697,A -85,B 0,C 180,E1 -19312.85,E2 -19312.85} C_VEL
LIN {X 0,Y 249.41,Z 279.353,A -85,B 0,C 180,E1 -19314.294,E2 -19314.294} C_VEL
LIN {X 0,Y 253.39,Z 291.496,A -85,B 0,C 180,E1 -19315.957,E2 -19315.957} C_VEL
LIN {X 0,Y 256.345,Z 303.452,A -85,B 0,C 180,E1 -19317.681,E2 -19317.681} C_VEL
LIN {X 0,Y 258.341,Z 315.549,A -85,B 0,C 180,E1 -19319.558,E2 -19319.558} C_VEL
LIN {X 0,Y 258.842,Z 321.281,A -85,B 0,C 180,E1 -19320.498,E2 -19320.498} C_VEL
LIN {X 0,Y 256.211,Z 332.847,A -85,B 0,C 180,E1 -19322.204,E2 -19322.204} C_VEL
LIN {X 0,Y 253.439,Z 343.337,A -85,B 0,C 180,E1 -19324.103,E2 -19324.103} C_VEL
LIN {X 0,Y 250.495,Z 353.752,A -85,B 0,C 180,E1 -19326.434,E2 -19326.434} C_VEL
LIN {X 0,Y 247.812,Z 362.341,A -85,B 0,C 180,E1 -19328.802,E2 -19328.802} C_VEL
LIN {X 0,Y 245.711,Z 369.258,A -85,B 0,C 180,E1 -19331.146,E2 -19331.146} C_VEL
LIN {X 0,Y 244.265,Z 374.497,A -85,B 0,C 180,E1 -19333.279,E2 -19333.279} C_VEL
LIN {X 0,Y 242.615,Z 379.573,A -85,B 0,C 180,E1 -19335.746,E2 -19335.746} C_VEL
LIN {X 0,Y 241.25,Z 384.825,A -85,B 0,C 180,E1 -19339.085,E2 -19339.085} C_VEL
LIN {X 0,Y 240.529,Z 387.756,A -85,B 0,C 180,E1 -19341.599,E2 -19341.599} C_VEL
LIN {X 0,Y 240.009,Z 390.445,A -85,B 0,C 180,E1 -19344.96,E2 -19344.96} C_VEL
LIN {X 0,Y 239.83,Z 391.788,A -85,B 0,C 180,E1 -19348.321,E2 -19348.321} C_VEL
LIN {X 0,Y 239.83,Z 391.816,A -85,B 0,C 180,E1 -19351.679,E2 -19351.679} C_VEL
LIN {X 0,Y 239.99,Z 390.526,A -85,B 0,C 180,E1 -19355.04,E2 -19355.04} C_VEL
LIN {X 0,Y 240.528,Z 387.885,A -85,B 0,C 180,E1 -19358.401,E2 -19358.401} C_VEL
LIN {X 0,Y 241.524,Z 383.824,A -85,B 0,C 180,E1 -19361.753,E2 -19361.753} C_VEL
LIN {X 0,Y 243.047,Z 378.212,A -85,B 0,C 180,E1 -19365.085,E2 -19365.085} C_VEL
LIN {X 0,Y 245.121,Z 371.868,A -85,B 0,C 180,E1 -19367.952,E2 -19367.952} C_VEL
LIN {X 0,Y 246.961,Z 365.211,A -85,B 0,C 180,E1 -19370.403,E2 -19370.403} C_VEL
LIN {X 0,Y 249.47,Z 357.209,A -85,B 0,C 180,E1 -19372.791,E2 -19372.791} C_VEL
LIN {X 0,Y 252.293,Z 347.556,A -85,B 0,C 180,E1 -19375.139,E2 -19375.139} C_VEL
LIN {X 0,Y 255.282,Z 336.837,A -85,B 0,C 180,E1 -19377.239,E2 -19377.239} C_VEL
LIN {X 0,Y 258.205,Z 324.956,A -85,B 0,C 180,E1 -19379.113,E2 -19379.113} C_VEL
LIN {X 0,Y 258.921,Z 320.772,A -85,B 0,C 180,E1 -19379.704,E2 -19379.704} C_VEL
LIN {X 0,Y 257.558,Z 309.744,A -85,B 0,C 180,E1 -19381.491,E2 -19381.491} C_VEL
LIN {X 0,Y 255.172,Z 298.025,A -85,B 0,C 180,E1 -19383.247,E2 -19383.247} C_VEL
LIN {X 0,Y 252.254,Z 287.634,A -85,B 0,C 180,E1 -19384.722,E2 -19384.722} C_VEL
LIN {X 0,Y 248.562,Z 277.195,A -85,B 0,C 180,E1 -19386.139,E2 -19386.139} C_VEL
LIN {X 0,Y 244.044,Z 266.705,A -85,B 0,C 180,E1 -19387.556,E2 -19387.556} C_VEL
LIN {X 0,Y 242.595,Z 263.524,A -85,B 0,C 180,E1 -19387.96,E2 -19387.96} C_VEL
LIN {X 0,Y 242.457,Z 262.766,A -85,B 0,C 180,E1 -19388.077,E2 -19388.077} C_VEL
LIN {X 0,Y 242.471,Z 260.138,A -85,B 0,C 180,E1 -19391.81,E2 -19391.81} C_VEL
LIN {X 0,Y 242.154,Z 257.524,A -85,B 0,C 180,E1 -19395.849,E2 -19395.849} C_VEL
LIN {X 0,Y 241.935,Z 256.178,A -85,B 0,C 180,E1 -19398.077,E2 -19398.077} C_VEL
LIN {X 0,Y 241.985,Z 255.969,A -85,B 0,C 180,E1 -19402.417,E2 -19402.417} C_VEL
LIN {X 0,Y 241.983,Z 255.968,A -85,B 0,C 180,E1 -19406.507,E2 -19406.507} C_VEL
LIN {X 0,Y 242.039,Z 255.961,A -85,B 0,C 180,E1 -19410.587,E2 -19410.587} C_VEL
LIN {X 0,Y 242.07,Z 255.953,A -85,B 0,C 180,E1 -19414.183,E2 -19414.183} C_VEL
LIN {X 0,Y 242.029,Z 255.962,A -85,B 0,C 180,E1 -19418.313,E2 -19418.313} C_VEL
LIN {X 0,Y 242.166,Z 255.945,A -85,B 0,C 180,E1 -19423.278,E2 -19423.278} C_VEL
LIN {X 0,Y 242.183,Z 255.944,A -85,B 0,C 180,E1 -19428.279,E2 -19428.279} C_VEL
LIN {X 0,Y 242.396,Z 255.915,A -85,B 0,C 180,E1 -19431.664,E2 -19431.664} C_VEL
LIN {X 0,Y 242.252,Z 255.933,A -85,B 0,C 180,E1 -19435.007,E2 -19435.007} C_VEL
LIN {X 0,Y 242.633,Z 255.887,A -85,B 0,C 180,E1 -19438.34,E2 -19438.34} C_VEL
LIN {X 0,Y 242.638,Z 255.886,A -85,B 0,C 180,E1 -19441.66,E2 -19441.66} C_VEL
LIN {X 0,Y 242.406,Z 255.915,A -85,B 0,C 180,E1 -19446.659,E2 -19446.659} C_VEL
LIN {X 0,Y 242.268,Z 255.932,A -85,B 0,C 180,E1 -19450.024,E2 -19450.024} C_VEL
LIN {X 0,Y 242.139,Z 255.95,A -85,B 0,C 180,E1 -19455.142,E2 -19455.142} C_VEL
LIN {X 0,Y 242.056,Z 255.958,A -85,B 0,C 180,E1 -19458.625,E2 -19458.625} C_VEL
LIN {X 0,Y 242.005,Z 255.966,A -85,B 0,C 180,E1 -19462.181,E2 -19462.181} C_VEL
LIN {X 0,Y 242.034,Z 255.954,A -85,B 0,C 180,E1 -19465.821,E2 -19465.821} C_VEL
LIN {X 0,Y 241.97,Z 255.969,A -85,B 0,C 180,E1 -19469.588,E2 -19469.588} C_VEL
LIN {X 0,Y 241.981,Z 255.967,A -85,B 0,C 180,E1 -19473.492,E2 -19473.492} C_VEL
LIN {X 0,Y 242.111,Z 256.694,A -85,B 0,C 180,E1 -19475.631,E2 -19475.631} C_VEL
LIN {X 0,Y 242.197,Z 257.303,A -85,B 0,C 180,E1 -19476.548,E2 -19476.548} C_VEL
LIN {X 0,Y 241.71,Z 258.356,A -85,B 0,C 180,E1 -19477.917,E2 -19477.917} C_VEL
LIN {X 0,Y 239.137,Z 260.446,A -85,B 0,C 180,E1 -19480.145,E2 -19480.145} C_VEL
LIN {X 0,Y 236.931,Z 262.189,A -85,B 0,C 180,E1 -19481.956,E2 -19481.956} C_VEL
LIN {X 0,Y 236.058,Z 263.408,A -85,B 0,C 180,E1 -19483.359,E2 -19483.359} C_VEL
LIN {X 0,Y 236.03,Z 263.781,A -85,B 0,C 180,E1 -19483.835,E2 -19483.835} C_VEL
LIN {X 0,Y 236.33,Z 266.142,A -85,B 0,C 180,E1 -19486.845,E2 -19486.845} C_VEL
LIN {X 0,Y 236.335,Z 269.555,A -85,B 0,C 180,E1 -19490.844,E2 -19490.844} C_VEL
LIN {X 0,Y 237.41,Z 272.806,A -85,B 0,C 180,E1 -19491.2,E2 -19491.2} C_VEL
LIN {X 0,Y 238.444,Z 274.923,A -85,B 0,C 180,E1 -19491.498,E2 -19491.498} C_VEL
LIN {X 0,Y 242.598,Z 285.819,A -85,B 0,C 180,E1 -19492.952,E2 -19492.952} C_VEL
LIN {X 0,Y 246.054,Z 297.183,A -85,B 0,C 180,E1 -19494.493,E2 -19494.493} C_VEL
LIN {X 0,Y 248.587,Z 308.736,A -85,B 0,C 180,E1 -19496.111,E2 -19496.111} C_VEL
LIN {X 0,Y 250.178,Z 320.719,A -85,B 0,C 180,E1 -19497.899,E2 -19497.899} C_VEL
LIN {X 0,Y 250.939,Z 331.782,A -85,B 0,C 180,E1 -19499.727,E2 -19499.727} C_VEL
LIN {X 0,Y 250.518,Z 335.801,A -85,B 0,C 180,E1 -19500.385,E2 -19500.385} C_VEL
LIN {X 0,Y 247.602,Z 347.229,A -85,B 0,C 180,E1 -19502.303,E2 -19502.303} C_VEL
LIN {X 0,Y 244.439,Z 357.677,A -85,B 0,C 180,E1 -19504.451,E2 -19504.451} C_VEL
LIN {X 0,Y 241.581,Z 367.123,A -85,B 0,C 180,E1 -19506.875,E2 -19506.875} C_VEL
LIN {X 0,Y 238.799,Z 376.123,A -85,B 0,C 180,E1 -19509.768,E2 -19509.768} C_VEL
LIN {X 0,Y 236.638,Z 383.401,A -85,B 0,C 180,E1 -19512.723,E2 -19512.723} C_VEL
LIN {X 0,Y 235.121,Z 388.504,A -85,B 0,C 180,E1 -19515.281,E2 -19515.281} C_VEL
LIN {X 0,Y 233.692,Z 393.771,A -85,B 0,C 180,E1 -19518.727,E2 -19518.727} C_VEL
LIN {X 0,Y 233.088,Z 396.726,A -85,B 0,C 180,E1 -19521.329,E2 -19521.329} C_VEL
LIN {X 0,Y 232.728,Z 399.431,A -85,B 0,C 180,E1 -19524.802,E2 -19524.802} C_VEL
LIN {X 0,Y 232.667,Z 400.77,A -85,B 0,C 180,E1 -19528.269,E2 -19528.269} C_VEL
LIN {X 0,Y 232.743,Z 400.935,A -85,B 0,C 180,E1 -19530,E2 -19530} C_VEL
LIN {X 0,Y 232.632,Z 400.253,A -85,B 0,C 180,E1 -19533.464,E2 -19533.464} C_VEL
LIN {X 0,Y 232.817,Z 398.223,A -85,B 0,C 180,E1 -19536.935,E2 -19536.935} C_VEL
LIN {X 0,Y 233.457,Z 394.798,A -85,B 0,C 180,E1 -19540.406,E2 -19540.406} C_VEL
LIN {X 0,Y 234.636,Z 389.876,A -85,B 0,C 180,E1 -19543.864,E2 -19543.864} C_VEL
LIN {X 0,Y 236.071,Z 385.135,A -85,B 0,C 180,E1 -19546.429,E2 -19546.429} C_VEL
LIN {X 0,Y 238.067,Z 378.261,A -85,B 0,C 180,E1 -19549.397,E2 -19549.397} C_VEL
LIN {X 0,Y 240.715,Z 369.735,A -85,B 0,C 180,E1 -19552.306,E2 -19552.306} C_VEL
LIN {X 0,Y 243.437,Z 360.842,A -85,B 0,C 180,E1 -19554.747,E2 -19554.747} C_VEL
LIN {X 0,Y 246.68,Z 350.075,A -85,B 0,C 180,E1 -19557.119,E2 -19557.119} C_VEL
LIN {X 0,Y 249.858,Z 338.399,A -85,B 0,C 180,E1 -19559.178,E2 -19559.178} C_VEL
LIN {X 0,Y 250.846,Z 333.731,A -85,B 0,C 180,E1 -19559.898,E2 -19559.898} C_VEL
LIN {X 0,Y 250.372,Z 322.963,A -85,B 0,C 180,E1 -19561.694,E2 -19561.694} C_VEL
LIN {X 0,Y 248.711,Z 309.62,A -85,B 0,C 180,E1 -19563.712,E2 -19563.712} C_VEL
LIN {X 0,Y 245.969,Z 297.077,A -85,B 0,C 180,E1 -19565.478,E2 -19565.478} C_VEL
LIN {X 0,Y 242.194,Z 284.722,A -85,B 0,C 180,E1 -19567.141,E2 -19567.141} C_VEL
LIN {X 0,Y 237.749,Z 273.427,A -85,B 0,C 180,E1 -19568.646,E2 -19568.646} C_VEL
LIN {X 0,Y 236.498,Z 270.59,A -85,B 0,C 180,E1 -19569.017,E2 -19569.017} C_VEL
LIN {X 0,Y 236.283,Z 269.408,A -85,B 0,C 180,E1 -19569.198,E2 -19569.198} C_VEL
LIN {X 0,Y 236.369,Z 267.051,A -85,B 0,C 180,E1 -19571.984,E2 -19571.984} C_VEL
LIN {X 0,Y 236.062,Z 264.162,A -85,B 0,C 180,E1 -19575.604,E2 -19575.604} C_VEL
LIN {X 0,Y 235.698,Z 261.617,A -85,B 0,C 180,E1 -19579.005,E2 -19579.005} C_VEL
LIN {X 0,Y 235.241,Z 258.693,A -85,B 0,C 180,E1 -19583.308,E2 -19583.308} C_VEL
LIN {X 0,Y 234.998,Z 257.393,A -85,B 0,C 180,E1 -19585.373,E2 -19585.373} C_VEL
LIN {X 0,Y 234.953,Z 256.847,A -85,B 0,C 180,E1 -19587.424,E2 -19587.424} C_VEL
LIN {X 0,Y 234.902,Z 256.851,A -85,B 0,C 180,E1 -19591.4,E2 -19591.4} C_VEL
LIN {X 0,Y 234.954,Z 256.845,A -85,B 0,C 180,E1 -19595.243,E2 -19595.243} C_VEL
LIN {X 0,Y 234.991,Z 256.84,A -85,B 0,C 180,E1 -19598.968,E2 -19598.968} C_VEL
LIN {X 0,Y 235.057,Z 256.829,A -85,B 0,C 180,E1 -19603.092,E2 -19603.092} C_VEL
LIN {X 0,Y 235.111,Z 256.824,A -85,B 0,C 180,E1 -19607.922,E2 -19607.922} C_VEL
LIN {X 0,Y 235.32,Z 256.798,A -85,B 0,C 180,E1 -19611.412,E2 -19611.412} C_VEL
LIN {X 0,Y 235.357,Z 256.792,A -85,B 0,C 180,E1 -19613.14,E2 -19613.14} C_VEL
LIN {X 0,Y 235.595,Z 256.765,A -85,B 0,C 180,E1 -19618.291,E2 -19618.291} C_VEL
LIN {X 0,Y 235.594,Z 256.762,A -85,B 0,C 180,E1 -19621.71,E2 -19621.71} C_VEL
LIN {X 0,Y 235.374,Z 256.79,A -85,B 0,C 180,E1 -19626.86,E2 -19626.86} C_VEL
LIN {X 0,Y 235.216,Z 256.811,A -85,B 0,C 180,E1 -19630.328,E2 -19630.328} C_VEL
LIN {X 0,Y 235.115,Z 256.823,A -85,B 0,C 180,E1 -19635.606,E2 -19635.606} C_VEL
LIN {X 0,Y 235.01,Z 256.838,A -85,B 0,C 180,E1 -19639.206,E2 -19639.206} C_VEL
LIN {X 0,Y 234.954,Z 256.844,A -85,B 0,C 180,E1 -19642.884,E2 -19642.884} C_VEL
LIN {X 0,Y 234.969,Z 256.841,A -85,B 0,C 180,E1 -19646.658,E2 -19646.658} C_VEL
LIN {X 0,Y 234.923,Z 256.848,A -85,B 0,C 180,E1 -19650.569,E2 -19650.569} C_VEL
LIN {X 0,Y 234.927,Z 256.848,A -85,B 0,C 180,E1 -19654.639,E2 -19654.639} C_VEL
LIN {X 0,Y 234.912,Z 256.85,A -85,B 0,C 180,E1 -19658.935,E2 -19658.935} C_VEL
LIN {X 0,Y 234.927,Z 257.165,A -85,B 0,C 180,E1 -19661.592,E2 -19661.592} C_VEL
LIN {X 0,Y 235.324,Z 259.658,A -85,B 0,C 180,E1 -19665.788,E2 -19665.788} C_VEL
LIN {X 0,Y 235.512,Z 261.702,A -85,B 0,C 180,E1 -19668.966,E2 -19668.966} C_VEL
LIN {X 0,Y 235.478,Z 262.962,A -85,B 0,C 180,E1 -19670.789,E2 -19670.789} C_VEL
LIN {X 0,Y 236.635,Z 266.167,A -85,B 0,C 180,E1 -19671.172,E2 -19671.172} C_VEL
LIN {X 0,Y 237.856,Z 268.32,A -85,B 0,C 180,E1 -19671.517,E2 -19671.517} C_VEL
LIN {X 0,Y 242.483,Z 279.023,A -85,B 0,C 180,E1 -19673.072,E2 -19673.072} C_VEL
LIN {X 0,Y 245.957,Z 289.059,A -85,B 0,C 180,E1 -19674.525,E2 -19674.525} C_VEL
LIN {X 0,Y 249.184,Z 300.947,A -85,B 0,C 180,E1 -19676.306,E2 -19676.306} C_VEL
LIN {X 0,Y 251.263,Z 311.934,A -85,B 0,C 180,E1 -19678.041,E2 -19678.041} C_VEL
LIN {X 0,Y 252.383,Z 321.541,A -85,B 0,C 180,E1 -19679.683,E2 -19679.683} C_VEL
LIN {X 0,Y 251.992,Z 324.852,A -85,B 0,C 180,E1 -19680.189,E2 -19680.189} C_VEL
LIN {X 0,Y 249.059,Z 336.344,A -85,B 0,C 180,E1 -19682.022,E2 -19682.022} C_VEL
LIN {X 0,Y 245.972,Z 347.167,A -85,B 0,C 180,E1 -19684.168,E2 -19684.168} C_VEL
LIN {X 0,Y 242.98,Z 356.906,A -85,B 0,C 180,E1 -19686.565,E2 -19686.565} C_VEL
LIN {X 0,Y 240.377,Z 364.983,A -85,B 0,C 180,E1 -19689.013,E2 -19689.013} C_VEL
LIN {X 0,Y 238.39,Z 371.706,A -85,B 0,C 180,E1 -19691.523,E2 -19691.523} C_VEL
LIN {X 0,Y 236.231,Z 378.106,A -85,B 0,C 180,E1 -19694.469,E2 -19694.469} C_VEL
LIN {X 0,Y 234.586,Z 383.775,A -85,B 0,C 180,E1 -19697.895,E2 -19697.895} C_VEL
LIN {X 0,Y 233.489,Z 387.892,A -85,B 0,C 180,E1 -19701.344,E2 -19701.344} C_VEL
LIN {X 0,Y 232.924,Z 390.58,A -85,B 0,C 180,E1 -19704.807,E2 -19704.807} C_VEL
LIN {X 0,Y 232.747,Z 391.923,A -85,B 0,C 180,E1 -19708.27,E2 -19708.27} C_VEL
LIN {X 0,Y 232.747,Z 391.95,A -85,B 0,C 180,E1 -19711.731,E2 -19711.731} C_VEL
LIN {X 0,Y 232.914,Z 390.604,A -85,B 0,C 180,E1 -19715.282,E2 -19715.282} C_VEL
LIN {X 0,Y 233.487,Z 388.019,A -85,B 0,C 180,E1 -19718.656,E2 -19718.656} C_VEL
LIN {X 0,Y 234.551,Z 383.958,A -85,B 0,C 180,E1 -19722.108,E2 -19722.108} C_VEL
LIN {X 0,Y 236.193,Z 378.346,A -85,B 0,C 180,E1 -19725.533,E2 -19725.533} C_VEL
LIN {X 0,Y 238.318,Z 372.002,A -85,B 0,C 180,E1 -19728.483,E2 -19728.483} C_VEL
LIN {X 0,Y 240.304,Z 365.344,A -85,B 0,C 180,E1 -19730.994,E2 -19730.994} C_VEL
LIN {X 0,Y 242.935,Z 357.341,A -85,B 0,C 180,E1 -19733.44,E2 -19733.44} C_VEL
LIN {X 0,Y 245.885,Z 347.687,A -85,B 0,C 180,E1 -19735.842,E2 -19735.842} C_VEL
LIN {X 0,Y 248.7,Z 338.035,A -85,B 0,C 180,E1 -19737.793,E2 -19737.793} C_VEL
LIN {X 0,Y 251.494,Z 327.252,A -85,B 0,C 180,E1 -19739.581,E2 -19739.581} C_VEL
LIN {X 0,Y 252.471,Z 322.084,A -85,B 0,C 180,E1 -19740.351,E2 -19740.351} C_VEL
LIN {X 0,Y 251.179,Z 310.976,A -85,B 0,C 180,E1 -19742.238,E2 -19742.238} C_VEL
LIN {X 0,Y 248.959,Z 299.748,A -85,B 0,C 180,E1 -19744.016,E2 -19744.016} C_VEL
LIN {X 0,Y 245.56,Z 287.397,A -85,B 0,C 180,E1 -19745.848,E2 -19745.848} C_VEL
LIN {X 0,Y 240.674,Z 274.474,A -85,B 0,C 180,E1 -19747.732,E2 -19747.732} C_VEL
LIN {X 0,Y 237.165,Z 267.011,A -85,B 0,C 180,E1 -19748.837,E2 -19748.837} C_VEL
LIN {X 0,Y 235.744,Z 264.122,A -85,B 0,C 180,E1 -19749.25,E2 -19749.25} C_VEL
LIN {X 0,Y 235.492,Z 262.959,A -85,B 0,C 180,E1 -19749.37,E2 -19749.37} C_VEL
LIN {X 0,Y 235.494,Z 261.338,A -85,B 0,C 180,E1 -19751.747,E2 -19751.747} C_VEL
LIN {X 0,Y 235.175,Z 258.786,A -85,B 0,C 180,E1 -19755.826,E2 -19755.826} C_VEL
LIN {X 0,Y 234.884,Z 257.027,A -85,B 0,C 180,E1 -19758.832,E2 -19758.832} C_VEL
LIN {X 0,Y 234.919,Z 256.849,A -85,B 0,C 180,E1 -19761.079,E2 -19761.079} C_VEL
LIN {X 0,Y 234.928,Z 256.847,A -85,B 0,C 180,E1 -19765.361,E2 -19765.361} C_VEL
LIN {X 0,Y 234.934,Z 256.846,A -85,B 0,C 180,E1 -19769.432,E2 -19769.432} C_VEL
LIN {X 0,Y 234.997,Z 256.837,A -85,B 0,C 180,E1 -19773.794,E2 -19773.794} C_VEL
LIN {X 0,Y 235.001,Z 256.839,A -85,B 0,C 180,E1 -19778.969,E2 -19778.969} C_VEL
LIN {X 0,Y 235.099,Z 256.826,A -85,B 0,C 180,E1 -19783.059,E2 -19783.059} C_VEL
LIN {X 0,Y 235.117,Z 256.823,A -85,B 0,C 180,E1 -19787.922,E2 -19787.922} C_VEL
LIN {X 0,Y 235.329,Z 256.796,A -85,B 0,C 180,E1 -19791.412,E2 -19791.412} C_VEL
LIN {X 0,Y 235.37,Z 256.792,A -85,B 0,C 180,E1 -19793.14,E2 -19793.14} C_VEL
LIN {X 0,Y 235.593,Z 256.764,A -85,B 0,C 180,E1 -19798.29,E2 -19798.29} C_VEL
LIN {X 0,Y 235.597,Z 256.763,A -85,B 0,C 180,E1 -19801.709,E2 -19801.709} C_VEL
LIN {X 0,Y 235.358,Z 256.792,A -85,B 0,C 180,E1 -19806.86,E2 -19806.86} C_VEL
LIN {X 0,Y 235.214,Z 256.811,A -85,B 0,C 180,E1 -19810.327,E2 -19810.327} C_VEL
LIN {X 0,Y 235.083,Z 256.829,A -85,B 0,C 180,E1 -19815.608,E2 -19815.608} C_VEL
LIN {X 0,Y 234.995,Z 256.838,A -85,B 0,C 180,E1 -19819.207,E2 -19819.207} C_VEL
LIN {X 0,Y 234.948,Z 256.843,A -85,B 0,C 180,E1 -19822.884,E2 -19822.884} C_VEL
LIN {X 0,Y 234.947,Z 256.84,A -85,B 0,C 180,E1 -19826.66,E2 -19826.66} C_VEL
LIN {X 0,Y 234.9,Z 256.85,A -85,B 0,C 180,E1 -19830.572,E2 -19830.572} C_VEL
LIN {X 0,Y 234.942,Z 256.845,A -85,B 0,C 180,E1 -19833.114,E2 -19833.114} C_VEL
LIN {X 0,Y 235.207,Z 258.449,A -85,B 0,C 180,E1 -19836.219,E2 -19836.219} C_VEL
LIN {X 0,Y 235.545,Z 260.385,A -85,B 0,C 180,E1 -19839.125,E2 -19839.125} C_VEL
LIN {X 0,Y 236.03,Z 263.781,A -85,B 0,C 180,E1 -19843.835,E2 -19843.835} C_VEL
LIN {X 0,Y 235.454,Z 264.608,A -85,B 0,C 180,E1 -19844.764,E2 -19844.764} C_VEL
LIN {X 0,Y 232.747,Z 266.212,A -85,B 0,C 180,E1 -19846.216,E2 -19846.216} C_VEL
LIN {X 0,Y 229.978,Z 267.849,A -85,B 0,C 180,E1 -19847.7,E2 -19847.7} C_VEL
LIN {X 0,Y 229.35,Z 268.73,A -85,B 0,C 180,E1 -19848.665,E2 -19848.665} C_VEL
LIN {X 0,Y 229.346,Z 269.379,A -85,B 0,C 180,E1 -19849.406,E2 -19849.406} C_VEL
LIN {X 0,Y 230.38,Z 272.509,A -85,B 0,C 180,E1 -19849.773,E2 -19849.773} C_VEL
LIN {X 0,Y 231.642,Z 274.765,A -85,B 0,C 180,E1 -19850.146,E2 -19850.146} C_VEL
LIN {X 0,Y 236.126,Z 286.098,A -85,B 0,C 180,E1 -19851.788,E2 -19851.788} C_VEL
LIN {X 0,Y 239.572,Z 297.498,A -85,B 0,C 180,E1 -19853.425,E2 -19853.425} C_VEL
LIN {X 0,Y 242.207,Z 309.418,A -85,B 0,C 180,E1 -19855.195,E2 -19855.195} C_VEL
LIN {X 0,Y 243.675,Z 320.559,A -85,B 0,C 180,E1 -19856.932,E2 -19856.932} C_VEL
LIN {X 0,Y 244.457,Z 331.643,A -85,B 0,C 180,E1 -19858.836,E2 -19858.836} C_VEL
LIN {X 0,Y 244.292,Z 335.763,A -85,B 0,C 180,E1 -19859.569,E2 -19859.569} C_VEL
LIN {X 0,Y 241.326,Z 347.098,A -85,B 0,C 180,E1 -19861.518,E2 -19861.518} C_VEL
LIN {X 0,Y 238.029,Z 357.544,A -85,B 0,C 180,E1 -19863.711,E2 -19863.711} C_VEL
LIN {X 0,Y 235.038,Z 366.99,A -85,B 0,C 180,E1 -19866.192,E2 -19866.192} C_VEL
LIN {X 0,Y 232.089,Z 375.989,A -85,B 0,C 180,E1 -19869.157,E2 -19869.157} C_VEL
LIN {X 0,Y 229.833,Z 383.267,A -85,B 0,C 180,E1 -19872.194,E2 -19872.194} C_VEL
LIN {X 0,Y 227.731,Z 389.808,A -85,B 0,C 180,E1 -19875.706,E2 -19875.706} C_VEL
LIN {X 0,Y 226.458,Z 394.708,A -85,B 0,C 180,E1 -19879.268,E2 -19879.268} C_VEL
LIN {X 0,Y 225.764,Z 398.117,A -85,B 0,C 180,E1 -19882.847,E2 -19882.847} C_VEL
LIN {X 0,Y 225.541,Z 400.134,A -85,B 0,C 180,E1 -19886.427,E2 -19886.427} C_VEL
LIN {X 0,Y 225.658,Z 400.801,A -85,B 0,C 180,E1 -19890,E2 -19890} C_VEL
LIN {X 0,Y 225.533,Z 400.118,A -85,B 0,C 180,E1 -19893.573,E2 -19893.573} C_VEL
LIN {X 0,Y 225.763,Z 398.088,A -85,B 0,C 180,E1 -19897.153,E2 -19897.153} C_VEL
LIN {X 0,Y 226.448,Z 394.662,A -85,B 0,C 180,E1 -19900.732,E2 -19900.732} C_VEL
LIN {X 0,Y 227.725,Z 389.739,A -85,B 0,C 180,E1 -19904.294,E2 -19904.294} C_VEL
LIN {X 0,Y 229.824,Z 383.181,A -85,B 0,C 180,E1 -19907.806,E2 -19907.806} C_VEL
LIN {X 0,Y 232.047,Z 375.882,A -85,B 0,C 180,E1 -19910.847,E2 -19910.847} C_VEL
LIN {X 0,Y 235.018,Z 366.847,A -85,B 0,C 180,E1 -19913.81,E2 -19913.81} C_VEL
LIN {X 0,Y 238.014,Z 357.371,A -85,B 0,C 180,E1 -19916.29,E2 -19916.29} C_VEL
LIN {X 0,Y 241.32,Z 346.887,A -85,B 0,C 180,E1 -19918.482,E2 -19918.482} C_VEL
LIN {X 0,Y 244.351,Z 335.346,A -85,B 0,C 180,E1 -19920.453,E2 -19920.453} C_VEL
LIN {X 0,Y 244.068,Z 325.099,A -85,B 0,C 180,E1 -19922.262,E2 -19922.262} C_VEL
LIN {X 0,Y 242.65,Z 312.1,A -85,B 0,C 180,E1 -19924.342,E2 -19924.342} C_VEL
LIN {X 0,Y 240.291,Z 300.442,A -85,B 0,C 180,E1 -19926.1,E2 -19926.1} C_VEL
LIN {X 0,Y 236.758,Z 288.061,A -85,B 0,C 180,E1 -19927.886,E2 -19927.886} C_VEL
LIN {X 0,Y 232.843,Z 277.652,A -85,B 0,C 180,E1 -19929.369,E2 -19929.369} C_VEL
LIN {X 0,Y 230.772,Z 273.189,A -85,B 0,C 180,E1 -19930.048,E2 -19930.048} C_VEL
LIN {X 0,Y 229.448,Z 270.06,A -85,B 0,C 180,E1 -19930.474,E2 -19930.474} C_VEL
LIN {X 0,Y 229.327,Z 269.291,A -85,B 0,C 180,E1 -19930.594,E2 -19930.594} C_VEL
LIN {X 0,Y 229.301,Z 267.628,A -85,B 0,C 180,E1 -19932.643,E2 -19932.643} C_VEL
LIN {X 0,Y 229.104,Z 265.704,A -85,B 0,C 180,E1 -19935.126,E2 -19935.126} C_VEL
LIN {X 0,Y 228.88,Z 263.938,A -85,B 0,C 180,E1 -19937.505,E2 -19937.505} C_VEL
LIN {X 0,Y 228.38,Z 260.881,A -85,B 0,C 180,E1 -19942.014,E2 -19942.014} C_VEL
LIN {X 0,Y 227.947,Z 258.197,A -85,B 0,C 180,E1 -19946.352,E2 -19946.352} C_VEL
LIN {X 0,Y 227.874,Z 257.726,A -85,B 0,C 180,E1 -19949.719,E2 -19949.719} C_VEL
LIN {X 0,Y 227.903,Z 257.722,A -85,B 0,C 180,E1 -19954.423,E2 -19954.423} C_VEL
LIN {X 0,Y 227.953,Z 257.716,A -85,B 0,C 180,E1 -19958.286,E2 -19958.286} C_VEL
LIN {X 0,Y 228.025,Z 257.708,A -85,B 0,C 180,E1 -19963.896,E2 -19963.896} C_VEL
LIN {X 0,Y 228.067,Z 257.702,A -85,B 0,C 180,E1 -19967.543,E2 -19967.543} C_VEL
LIN {X 0,Y 228.259,Z 257.677,A -85,B 0,C 180,E1 -19971.144,E2 -19971.144} C_VEL
LIN {X 0,Y 228.309,Z 257.67,A -85,B 0,C 180,E1 -19972.927,E2 -19972.927} C_VEL
LIN {X 0,Y 228.554,Z 257.642,A -85,B 0,C 180,E1 -19978.238,E2 -19978.238} C_VEL
LIN {X 0,Y 228.553,Z 257.639,A -85,B 0,C 180,E1 -19981.762,E2 -19981.762} C_VEL
LIN {X 0,Y 228.325,Z 257.668,A -85,B 0,C 180,E1 -19987.073,E2 -19987.073} C_VEL
LIN {X 0,Y 228.147,Z 257.691,A -85,B 0,C 180,E1 -19990.651,E2 -19990.651} C_VEL
LIN {X 0,Y 228.067,Z 257.7,A -85,B 0,C 180,E1 -19994.272,E2 -19994.272} C_VEL
LIN {X 0,Y 228.005,Z 257.708,A -85,B 0,C 180,E1 -19997.953,E2 -19997.953} C_VEL
LIN {X 0,Y 227.918,Z 257.718,A -85,B 0,C 180,E1 -20002.321,E2 -20002.321} C_VEL
LIN {X 0,Y 227.943,Z 257.716,A -85,B 0,C 180,E1 -20006.602,E2 -20006.602} C_VEL
LIN {X 0,Y 227.898,Z 257.722,A -85,B 0,C 180,E1 -20010.291,E2 -20010.291} C_VEL
LIN {X 0,Y 227.878,Z 257.726,A -85,B 0,C 180,E1 -20013.721,E2 -20013.721} C_VEL
LIN {X 0,Y 227.84,Z 257.73,A -85,B 0,C 180,E1 -20018.092,E2 -20018.092} C_VEL
LIN {X 0,Y 227.813,Z 257.803,A -85,B 0,C 180,E1 -20020.38,E2 -20020.38} C_VEL
